C01810=1043.766,333.386,381.693,172.543,41.628,158.015
C01811=1043.756,333.058,381.740,172.537,41.623,158.014
C01812=1043.749,332.811,381.775,172.532,41.620,158.013
C01813=1043.742,332.564,381.811,172.528,41.617,158.012
C01814=1043.736,332.315,381.847,172.522,41.614,158.011
C01815=1043.728,332.069,381.883,172.518,41.611,158.010
C01816=1043.721,331.821,381.919,172.514,41.608,158.009
C01817=1043.714,331.573,381.954,172.509,41.605,158.008
C01818=1043.707,331.326,381.990,172.505,41.602,158.007
C01819=1043.700,331.078,382.025,172.500,41.599,158.006
C01820=1043.693,330.832,382.061,172.495,41.595,158.005
C01821=1043.686,330.584,382.096,172.491,41.592,158.004
C01822=1043.679,330.336,382.132,172.486,41.589,158.003
C01823=1043.672,330.090,382.167,172.482,41.586,158.002
C01824=1043.665,329.842,382.203,172.478,41.583,158.001
C01825=1043.657,329.594,382.238,172.473,41.580,158.000
C01826=1043.650,329.347,382.274,172.469,41.577,157.999
C01827=1043.643,329.100,382.308,172.465,41.573,157.998
C01828=1043.635,328.852,382.344,172.459,41.570,157.997
C01829=1043.629,328.605,382.379,172.456,41.568,157.996
C01830=1043.621,328.358,382.414,172.450,41.565,157.995
C01831=1043.614,328.110,382.449,172.446,41.562,157.994
C01832=1043.607,327.862,382.484,172.442,41.558,157.993
C01833=1043.600,327.615,382.519,172.437,41.556,157.993
C01834=1043.592,327.367,382.554,172.433,41.553,157.992
C01835=1043.585,327.120,382.589,172.429,41.550,157.991
C01836=1043.578,326.873,382.624,172.424,41.547,157.990
C01837=1043.571,326.625,382.659,172.420,41.544,157.989
C01838=1043.563,326.378,382.694,172.416,41.541,157.988
C01839=1043.556,326.130,382.729,172.411,41.538,157.987
C01840=1043.549,325.883,382.764,172.407,41.535,157.986
C01841=1043.541,325.635,382.799,172.403,41.532,157.985
C01842=1043.534,325.388,382.834,172.398,41.529,157.984
C01843=1043.527,325.141,382.869,172.393,41.526,157.983
C01844=1043.520,324.893,382.904,172.389,41.524,157.982
C01845=1043.513,324.646,382.939,172.384,41.521,157.981
C01846=1043.506,324.398,382.973,172.380,41.517,157.980
C01847=1043.498,324.151,383.008,172.376,41.515,157.980
C01848=1043.492,323.903,383.043,172.372,41.512,157.979
C01849=1043.485,323.656,383.078,172.367,41.509,157.978
C01850=1043.477,323.409,383.113,172.363,41.506,157.977
C01851=1043.471,323.161,383.147,172.359,41.503,157.976
C01852=1043.463,322.914,383.182,172.355,41.500,157.975
C01853=1043.456,322.666,383.217,172.350,41.497,157.974
C01854=1043.449,322.418,383.251,172.346,41.494,157.973
C01855=1043.442,322.171,383.286,172.342,41.492,157.972
C01856=1043.434,321.924,383.321,172.338,41.488,157.971
C01857=1043.428,321.676,383.355,172.333,41.486,157.970
C01858=1043.420,321.429,383.390,172.329,41.483,157.969
C01859=1043.414,321.181,383.425,172.325,41.480,157.969
C01860=1043.407,320.933,383.459,172.321,41.477,157.968
C01861=1043.400,320.686,383.494,172.317,41.474,157.967
C01862=1043.393,320.438,383.528,172.312,41.471,157.966
C01863=1043.386,320.191,383.563,172.308,41.469,157.965
C01864=1043.376,319.858,383.609,172.302,41.465,157.964
C01865=1043.367,319.524,383.656,172.297,41.461,157.963
C01866=1043.358,319.191,383.702,172.291,41.457,157.962
C01867=1043.348,318.858,383.749,172.285,41.453,157.960
C01868=1043.342,318.611,383.782,172.281,41.451,157.959
C01869=1043.335,318.363,383.817,172.277,41.447,157.958
C01870=1043.328,318.116,383.851,172.273,41.445,157.958
C01871=1043.321,317.868,383.886,172.268,41.442,157.957
C01872=1043.314,317.621,383.920,172.264,41.439,157.956
C01873=1043.307,317.373,383.955,172.260,41.437,157.955
C01874=1043.300,317.126,383.989,172.256,41.433,157.954
C01875=1043.293,316.878,384.024,172.252,41.431,157.953
C01876=1043.286,316.630,384.057,172.248,41.428,157.952
C01877=1043.280,316.383,384.091,172.244,41.425,157.952
C01878=1043.273,316.136,384.126,172.240,41.423,157.951
C01879=1043.266,315.888,384.160,172.236,41.419,157.950
C01880=1043.259,315.640,384.194,172.231,41.417,157.949
C01881=1043.252,315.392,384.229,172.227,41.414,157.948
C01882=1043.245,315.145,384.263,172.223,41.411,157.947
C01883=1043.239,314.898,384.297,172.219,41.409,157.946
C01884=1043.232,314.650,384.331,172.215,41.406,157.946
C01885=1043.225,314.402,384.366,172.211,41.403,157.945
C01886=1043.218,314.154,384.399,172.207,41.400,157.944
C01887=1043.212,313.908,384.434,172.204,41.398,157.943
C01888=1043.205,313.660,384.468,172.200,41.395,157.942
C01889=1043.198,313.412,384.502,172.196,41.392,157.941
C01890=1043.191,313.164,384.536,172.192,41.389,157.940
C01891=1043.185,312.917,384.570,172.188,41.387,157.940
C01892=1043.178,312.669,384.604,172.184,41.383,157.939
C01893=1043.171,312.422,384.638,172.180,41.381,157.938
C01894=1043.164,312.175,384.671,172.176,41.378,157.937
C01895=1043.157,311.927,384.705,172.171,41.376,157.936
C01896=1043.150,311.679,384.739,172.167,41.373,157.935
C01897=1043.143,311.432,384.773,172.163,41.371,157.935
C01898=1043.136,311.183,384.806,172.159,41.368,157.934
C01899=1043.129,310.936,384.839,172.155,41.365,157.933
C01900=1043.122,310.689,384.873,172.151,41.363,157.932
C01901=1043.115,310.441,384.907,172.147,41.360,157.931
C01902=1043.108,310.193,384.940,172.143,41.358,157.931
C01903=1043.101,309.946,384.973,172.140,41.355,157.930
C01904=1043.093,309.698,385.007,172.136,41.352,157.929
C01905=1043.086,309.451,385.041,172.132,41.350,157.928
C01906=1043.080,309.203,385.073,172.128,41.348,157.927
C01907=1043.073,308.955,385.107,172.124,41.345,157.927
C01908=1043.066,308.708,385.141,172.120,41.343,157.926
C01909=1043.059,308.459,385.174,172.116,41.340,157.925
C01910=1043.052,308.212,385.208,172.112,41.337,157.924
C01911=1043.044,307.965,385.241,172.108,41.335,157.923
C01912=1043.038,307.718,385.274,172.105,41.332,157.923
C01913=1043.031,307.470,385.307,172.101,41.330,157.922
C01914=1043.024,307.222,385.341,172.097,41.327,157.921
C01915=1043.017,306.975,385.374,172.093,41.325,157.920
C01916=1043.010,306.726,385.407,172.089,41.322,157.920
C01917=1043.003,306.479,385.441,172.085,41.320,157.919
C01918=1042.996,306.232,385.474,172.081,41.317,157.918
C01919=1042.989,305.984,385.507,172.077,41.314,157.917
C01920=1042.980,305.655,385.551,172.072,41.311,157.916
C01921=1042.971,305.326,385.595,172.067,41.308,157.915
C01922=1042.962,304.998,385.639,172.062,41.305,157.914
C01923=1042.953,304.669,385.683,172.057,41.302,157.913
C01924=1042.946,304.422,385.716,172.053,41.299,157.912
C01925=1042.939,304.174,385.749,172.049,41.296,157.911
C01926=1042.933,303.926,385.782,172.045,41.294,157.911
C01927=1042.925,303.679,385.815,172.041,41.291,157.910
C01928=1042.919,303.431,385.848,172.038,41.289,157.909
C01929=1042.912,303.183,385.881,172.034,41.286,157.908
C01930=1042.905,302.936,385.915,172.030,41.284,157.908
C01931=1042.898,302.688,385.948,172.026,41.281,157.907
C01932=1042.892,302.440,385.981,172.023,41.279,157.906
C01933=1042.884,302.193,386.014,172.019,41.277,157.905
C01934=1042.878,301.945,386.046,172.015,41.274,157.905
C01935=1042.871,301.697,386.079,172.011,41.271,157.904
C01936=1042.864,301.449,386.112,172.008,41.269,157.903
C01937=1042.858,301.202,386.146,172.004,41.267,157.902
C01938=1042.850,300.954,386.178,172.000,41.264,157.902
C01939=1042.844,300.707,386.211,171.996,41.261,157.901
C01940=1042.838,300.459,386.244,171.992,41.259,157.900
C01941=1042.831,300.211,386.277,171.989,41.257,157.899
C01942=1042.824,299.963,386.310,171.985,41.254,157.899
C01943=1042.816,299.716,386.343,171.982,41.252,157.898
C01944=1042.810,299.468,386.376,171.978,41.249,157.897
C01945=1042.804,299.221,386.408,171.974,41.247,157.896
C01946=1042.797,298.972,386.441,171.970,41.244,157.895
C01947=1042.791,298.725,386.474,171.967,41.242,157.895
C01948=1042.784,298.477,386.506,171.963,41.239,157.894
C01949=1042.777,298.229,386.539,171.960,41.237,157.893
C01950=1042.770,297.981,386.572,171.956,41.235,157.893
C01951=1042.764,297.734,386.605,171.952,41.232,157.892
C01952=1042.758,297.486,386.638,171.948,41.229,157.891
C01953=1042.750,297.238,386.670,171.945,41.227,157.890
C01954=1042.744,296.991,386.703,171.941,41.225,157.890
C01955=1042.738,296.743,386.736,171.938,41.223,157.889
C01956=1042.731,296.496,386.768,171.934,41.220,157.888
C01957=1042.724,296.248,386.801,171.930,41.217,157.887
C01958=1042.717,296.000,386.834,171.927,41.215,157.887
C01959=1042.711,295.752,386.866,171.923,41.213,157.886
C01960=1042.705,295.504,386.898,171.919,41.210,157.885
C01961=1042.698,295.256,386.931,171.916,41.208,157.884
C01962=1042.691,295.009,386.963,171.913,41.206,157.884
C01963=1042.684,294.761,386.996,171.909,41.203,157.883
C01964=1042.678,294.513,387.027,171.905,41.201,157.882
C01965=1042.671,294.265,387.060,171.901,41.198,157.882
C01966=1042.664,294.018,387.093,171.898,41.196,157.881
C01967=1042.658,293.770,387.125,171.895,41.194,157.880
C01968=1042.651,293.522,387.157,171.891,41.192,157.879
C01969=1042.644,293.274,387.190,171.887,41.189,157.879
C01970=1042.637,293.026,387.221,171.884,41.187,157.878
C01971=1042.630,292.779,387.253,171.881,41.185,157.877
C01972=1042.624,292.531,387.286,171.877,41.182,157.877
C01973=1042.616,292.283,387.318,171.873,41.180,157.876
C01974=1042.609,292.035,387.350,171.869,41.177,157.875
C01975=1042.603,291.787,387.382,171.866,41.175,157.875
C01976=1042.594,291.475,387.423,171.862,41.173,157.874
C01977=1042.586,291.163,387.462,171.858,41.170,157.873
C01978=1042.578,290.851,387.503,171.853,41.167,157.872
C01979=1042.569,290.539,387.544,171.849,41.164,157.871
C01980=1042.562,290.290,387.576,171.845,41.162,157.870
C01981=1042.556,290.042,387.608,171.841,41.159,157.870
C01982=1042.549,289.795,387.640,171.837,41.157,157.869
C01983=1042.542,289.547,387.671,171.835,41.155,157.868
C01984=1042.535,289.300,387.703,171.831,41.153,157.868
C01985=1042.529,289.052,387.735,171.827,41.150,157.867
C01986=1042.522,288.804,387.767,171.824,41.148,157.866
C01987=1042.515,288.556,387.799,171.821,41.146,157.866
C01988=1042.508,288.308,387.831,171.817,41.143,157.865
C01989=1042.501,288.060,387.862,171.814,41.141,157.864
C01990=1042.495,287.812,387.895,171.810,41.139,157.864
C01991=1042.488,287.564,387.926,171.807,41.137,157.863
C01992=1042.482,287.316,387.958,171.803,41.135,157.862
C01993=1042.475,287.069,387.989,171.800,41.132,157.861
C01994=1042.468,286.821,388.021,171.796,41.130,157.861
C01995=1042.461,286.573,388.053,171.793,41.128,157.860
C01996=1042.454,286.325,388.084,171.790,41.126,157.860
C01997=1042.448,286.077,388.116,171.786,41.123,157.859
C01998=1042.442,285.829,388.148,171.782,41.121,157.858
C01999=1042.434,285.581,388.179,171.780,41.119,157.857
C02000=1042.427,285.333,388.212,171.776,41.117,157.857
C02001=1042.421,285.086,388.243,171.772,41.115,157.856
C02002=1042.414,284.838,388.275,171.770,41.113,157.856
C02003=1042.407,284.590,388.306,171.766,41.110,157.855
C02004=1042.400,284.342,388.337,171.762,41.108,157.854
C02005=1042.394,284.094,388.369,171.759,41.106,157.854
C02006=1042.387,283.846,388.400,171.755,41.104,157.853
C02007=1042.380,283.598,388.432,171.752,41.102,157.852
C02008=1042.373,283.350,388.463,171.749,41.100,157.852
C02009=1042.367,283.102,388.495,171.745,41.098,157.851
C02010=1042.360,282.854,388.526,171.743,41.096,157.850
C02011=1042.353,282.607,388.557,171.739,41.093,157.850
C02012=1042.347,282.359,388.589,171.735,41.091,157.849
C02013=1042.340,282.111,388.620,171.732,41.089,157.848
C02014=1042.333,281.863,388.652,171.729,41.087,157.848
C02015=1042.326,281.615,388.683,171.726,41.084,157.847
C02016=1042.320,281.366,388.714,171.722,41.082,157.846
C02017=1042.314,281.119,388.745,171.719,41.080,157.846
C02018=1042.307,280.871,388.776,171.716,41.078,157.845
C02019=1042.300,280.623,388.808,171.712,41.076,157.844
C02020=1042.294,280.376,388.839,171.709,41.073,157.844
C02021=1042.287,280.128,388.871,171.706,41.071,157.843
C02022=1042.280,279.880,388.902,171.702,41.069,157.842
C02023=1042.274,279.631,388.933,171.699,41.067,157.842
C02024=1042.267,279.383,388.964,171.695,41.065,157.841
C02025=1042.260,279.135,388.996,171.693,41.063,157.841
C02026=1042.254,278.888,389.027,171.689,41.061,157.840
C02027=1042.248,278.640,389.057,171.686,41.059,157.839
C02028=1042.240,278.392,389.088,171.683,41.057,157.839
C02029=1042.234,278.144,389.120,171.679,41.054,157.838
C02030=1042.227,277.896,389.150,171.676,41.052,157.837
C02031=1042.220,277.648,389.182,171.673,41.050,157.837
C02032=1042.212,277.348,389.219,171.669,41.048,157.836
C02033=1042.204,277.047,389.257,171.665,41.045,157.835
C02034=1042.196,276.747,389.294,171.661,41.043,157.834
C02035=1042.187,276.446,389.331,171.657,41.040,157.834
C02036=1042.181,276.198,389.363,171.654,41.038,157.833
C02037=1042.175,275.950,389.393,171.651,41.036,157.832
C02038=1042.168,275.702,389.425,171.647,41.034,157.832
C02039=1042.161,275.454,389.455,171.644,41.032,157.831
C02040=1042.154,275.206,389.486,171.641,41.030,157.831
C02041=1042.148,274.958,389.517,171.638,41.027,157.830
C02042=1042.142,274.710,389.548,171.634,41.025,157.829
C02043=1042.135,274.462,389.578,171.632,41.023,157.829
C02044=1042.128,274.214,389.609,171.628,41.021,157.828
C02045=1042.121,273.966,389.640,171.625,41.020,157.828
C02046=1042.114,273.718,389.671,171.622,41.017,157.827
C02047=1042.108,273.470,389.701,171.619,41.015,157.826
C02048=1042.101,273.223,389.732,171.615,41.013,157.826
C02049=1042.094,272.974,389.763,171.613,41.011,157.825
C02050=1042.088,272.726,389.794,171.609,41.009,157.824
C02051=1042.081,272.479,389.824,171.606,41.007,157.824
C02052=1042.075,272.230,389.855,171.603,41.005,157.823
C02053=1042.068,271.982,389.886,171.600,41.003,157.822
C02054=1042.061,271.734,389.916,171.596,41.001,157.822
C02055=1042.055,271.486,389.947,171.594,40.999,157.821
C02056=1042.049,271.238,389.977,171.591,40.997,157.821
C02057=1042.041,270.990,390.008,171.587,40.995,157.820
C02058=1042.035,270.742,390.039,171.585,40.992,157.819
C02059=1042.028,270.494,390.069,171.581,40.990,157.819
C02060=1042.022,270.246,390.099,171.578,40.989,157.818
C02061=1042.014,269.998,390.130,171.575,40.987,157.818
C02062=1042.009,269.750,390.160,171.572,40.984,157.817
C02063=1042.001,269.502,390.191,171.568,40.982,157.816
C02064=1041.995,269.254,390.222,171.566,40.980,157.816
C02065=1041.988,269.005,390.252,171.562,40.979,157.815
C02066=1041.982,268.758,390.282,171.559,40.977,157.815
C02067=1041.975,268.509,390.312,171.557,40.974,157.814
C02068=1041.968,268.261,390.342,171.553,40.972,157.813
C02069=1041.962,268.013,390.373,171.550,40.970,157.813
C02070=1041.955,267.765,390.403,171.547,40.969,157.812
C02071=1041.949,267.517,390.433,171.544,40.966,157.812
C02072=1041.942,267.269,390.463,171.540,40.964,157.811
C02073=1041.935,267.021,390.494,171.538,40.962,157.811
C02074=1041.929,266.773,390.524,171.535,40.961,157.810
C02075=1041.921,266.525,390.554,171.531,40.959,157.809
C02076=1041.915,266.276,390.585,171.529,40.956,157.809
C02077=1041.908,266.029,390.614,171.525,40.954,157.808
C02078=1041.901,265.781,390.644,171.523,40.953,157.808
C02079=1041.895,265.532,390.675,171.520,40.950,157.807
C02080=1041.888,265.285,390.705,171.516,40.948,157.806
C02081=1041.881,265.036,390.735,171.514,40.946,157.806
C02082=1041.875,264.788,390.765,171.510,40.945,157.805
C02083=1041.868,264.540,390.795,171.507,40.943,157.805
C02084=1041.861,264.292,390.826,171.505,40.940,157.804
C02085=1041.855,264.044,390.856,171.501,40.939,157.804
C02086=1041.848,263.795,390.885,171.498,40.937,157.803
C02087=1041.842,263.548,390.915,171.496,40.934,157.802
C02088=1041.833,263.252,390.952,171.492,40.932,157.802
C02089=1041.826,262.956,390.987,171.488,40.930,157.801
C02090=1041.818,262.660,391.023,171.484,40.928,157.800
C02091=1041.810,262.364,391.059,171.481,40.925,157.800
C02092=1041.803,262.116,391.088,171.478,40.923,157.799
C02093=1041.797,261.868,391.118,171.475,40.921,157.798
C02094=1041.790,261.620,391.148,171.472,40.920,157.798
C02095=1041.783,261.372,391.177,171.469,40.917,157.797
C02096=1041.776,261.123,391.207,171.466,40.916,157.797
C02097=1041.769,260.875,391.237,171.463,40.914,157.796
C02098=1041.763,260.627,391.267,171.461,40.912,157.796
C02099=1041.756,260.379,391.297,171.457,40.910,157.795
C02100=1041.750,260.131,391.326,171.454,40.908,157.794
C02101=1041.742,259.883,391.356,171.452,40.906,157.794
C02102=1041.736,259.634,391.385,171.448,40.904,157.793
C02103=1041.729,259.386,391.415,171.445,40.903,157.793
C02104=1041.723,259.138,391.444,171.443,40.900,157.792
C02105=1041.715,258.890,391.474,171.439,40.899,157.792
C02106=1041.708,258.641,391.503,171.437,40.897,157.791
C02107=1041.701,258.394,391.533,171.434,40.895,157.791
C02108=1041.695,258.145,391.562,171.430,40.893,157.790
C02109=1041.688,257.898,391.592,171.428,40.891,157.790
C02110=1041.681,257.649,391.621,171.425,40.889,157.789
C02111=1041.675,257.401,391.651,171.422,40.888,157.788
C02112=1041.668,257.153,391.680,171.419,40.886,157.788
C02113=1041.661,256.905,391.710,171.416,40.884,157.787
C02114=1041.655,256.657,391.739,171.413,40.882,157.787
C02115=1041.648,256.408,391.769,171.410,40.880,157.786
C02116=1041.642,256.160,391.798,171.408,40.878,157.786
C02117=1041.635,255.912,391.828,171.405,40.876,157.785
C02118=1041.627,255.664,391.857,171.401,40.874,157.785
C02119=1041.621,255.415,391.886,171.399,40.872,157.784
C02120=1041.614,255.167,391.915,171.396,40.871,157.784
C02121=1041.608,254.920,391.945,171.393,40.868,157.783
C02122=1041.601,254.671,391.975,171.390,40.867,157.782
C02123=1041.595,254.423,392.004,171.387,40.865,157.782
C02124=1041.587,254.175,392.034,171.385,40.863,157.781
C02125=1041.581,253.927,392.063,171.382,40.861,157.781
C02126=1041.575,253.678,392.092,171.379,40.859,157.780
C02127=1041.568,253.430,392.121,171.376,40.857,157.780
C02128=1041.562,253.182,392.151,171.373,40.855,157.779
C02129=1041.554,252.934,392.180,171.371,40.853,157.779
C02130=1041.548,252.685,392.209,171.367,40.852,157.778
C02131=1041.541,252.437,392.238,171.365,40.850,157.777
C02132=1041.535,252.188,392.267,171.362,40.847,157.777
C02133=1041.528,251.941,392.297,171.359,40.846,157.776
C02134=1041.522,251.693,392.326,171.356,40.844,157.776
C02135=1041.515,251.444,392.356,171.353,40.842,157.775
C02136=1041.509,251.196,392.385,171.350,40.840,157.775
C02137=1041.502,250.948,392.413,171.348,40.838,157.774
C02138=1041.495,250.701,392.443,171.345,40.836,157.774
C02139=1041.488,250.452,392.472,171.342,40.835,157.773
C02140=1041.482,250.204,392.501,171.339,40.832,157.772
C02141=1041.476,249.955,392.530,171.337,40.831,157.772
C02142=1041.469,249.707,392.560,171.334,40.828,157.771
C02143=1041.463,249.458,392.589,171.331,40.827,157.771
C02144=1041.455,249.161,392.624,171.328,40.824,157.770
C02145=1041.447,248.864,392.658,171.324,40.822,157.770
C02146=1041.439,248.567,392.693,171.321,40.820,157.769
C02147=1041.431,248.269,392.728,171.318,40.818,157.768
C02148=1041.425,248.021,392.757,171.315,40.816,157.768
C02149=1041.418,247.772,392.786,171.312,40.814,157.767
C02150=1041.412,247.524,392.815,171.310,40.812,157.767
C02151=1041.406,247.276,392.844,171.307,40.810,157.766
C02152=1041.399,247.028,392.873,171.304,40.808,157.766
C02153=1041.392,246.780,392.902,171.301,40.806,157.765
C02154=1041.386,246.531,392.931,171.298,40.804,157.764
C02155=1041.380,246.283,392.960,171.296,40.802,157.764
C02156=1041.373,246.035,392.989,171.293,40.800,157.763
C02157=1041.367,245.787,393.018,171.290,40.798,157.763
C02158=1041.360,245.539,393.047,171.288,40.796,157.762
C02159=1041.353,245.290,393.076,171.285,40.794,157.762
C02160=1041.347,245.042,393.104,171.283,40.793,157.761
C02161=1041.341,244.793,393.134,171.279,40.791,157.761
C02162=1041.334,244.546,393.162,171.277,40.789,157.760
C02163=1041.328,244.298,393.191,171.274,40.787,157.759
C02164=1041.320,244.049,393.220,171.271,40.785,157.759
C02165=1041.314,243.800,393.248,171.269,40.783,157.759
C02166=1041.308,243.552,393.277,171.266,40.781,157.758
C02167=1041.301,243.304,393.306,171.264,40.780,157.757
C02168=1041.295,243.056,393.335,171.261,40.777,157.757
C02169=1041.288,242.808,393.362,171.259,40.776,157.756
C02170=1041.281,242.559,393.392,171.255,40.774,157.756
C02171=1041.275,242.311,393.421,171.252,40.772,157.755
C02172=1041.268,242.062,393.449,171.250,40.770,157.755
C02173=1041.262,241.814,393.478,171.247,40.768,157.754
C02174=1041.255,241.566,393.506,171.245,40.767,157.754
C02175=1041.249,241.318,393.534,171.242,40.764,157.753
C02176=1041.242,241.070,393.563,171.240,40.763,157.753
C02177=1041.235,240.821,393.592,171.237,40.761,157.752
C02178=1041.229,240.573,393.620,171.234,40.759,157.752
C02179=1041.222,240.324,393.649,171.232,40.757,157.751
C02180=1041.216,240.076,393.677,171.229,40.755,157.751
C02181=1041.209,239.828,393.705,171.226,40.754,157.750
C02182=1041.203,239.579,393.734,171.223,40.752,157.750
C02183=1041.196,239.332,393.762,171.221,40.750,157.749
C02184=1041.188,239.082,393.790,171.218,40.748,157.749
C02185=1041.182,238.834,393.819,171.215,40.747,157.748
C02186=1041.176,238.586,393.847,171.213,40.744,157.747
C02187=1041.169,238.338,393.875,171.210,40.743,157.747
C02188=1041.163,238.089,393.904,171.208,40.741,157.747
C02189=1041.156,237.841,393.932,171.205,40.739,157.746
C02190=1041.149,237.593,393.960,171.203,40.737,157.745
C02191=1041.143,237.345,393.989,171.200,40.736,157.745
C02192=1041.136,237.096,394.017,171.197,40.733,157.744
C02193=1041.129,236.848,394.044,171.195,40.732,157.744
C02194=1041.122,236.600,394.073,171.192,40.730,157.743
C02195=1041.116,236.351,394.101,171.190,40.728,157.743
C02196=1041.109,236.103,394.130,171.187,40.726,157.742
C02197=1041.102,235.854,394.158,171.185,40.725,157.742
C02198=1041.095,235.606,394.185,171.181,40.723,157.741
C02199=1041.089,235.358,394.214,171.179,40.721,157.741
C02200=1041.081,235.054,394.248,171.176,40.719,157.740
C02201=1041.073,234.752,394.282,171.173,40.716,157.740
C02202=1041.065,234.449,394.316,171.170,40.714,157.739
C02203=1041.057,234.146,394.351,171.167,40.712,157.738
C02204=1041.051,233.897,394.379,171.164,40.710,157.738
C02205=1041.044,233.649,394.407,171.162,40.708,157.737
C02206=1041.037,233.401,394.435,171.159,40.707,157.737
C02207=1041.031,233.152,394.463,171.157,40.704,157.736
C02208=1041.025,232.904,394.491,171.154,40.703,157.736
C02209=1041.018,232.655,394.519,171.152,40.701,157.735
C02210=1041.011,232.407,394.548,171.149,40.699,157.735
C02211=1041.004,232.159,394.575,171.147,40.697,157.734
C02212=1040.998,231.910,394.604,171.144,40.696,157.734
C02213=1040.992,231.662,394.631,171.141,40.693,157.733
C02214=1040.985,231.413,394.659,171.139,40.692,157.733
C02215=1040.978,231.165,394.687,171.136,40.690,157.732
C02216=1040.972,230.916,394.714,171.134,40.688,157.732
C02217=1040.965,230.669,394.743,171.131,40.686,157.731
C02218=1040.958,230.420,394.771,171.129,40.685,157.731
C02219=1040.951,230.172,394.798,171.126,40.682,157.730
C02220=1040.945,229.923,394.826,171.124,40.681,157.730
C02221=1040.939,229.675,394.854,171.121,40.679,157.729
C02222=1040.932,229.426,394.882,171.118,40.677,157.729
C02223=1040.925,229.178,394.910,171.116,40.675,157.728
C02224=1040.919,228.929,394.938,171.113,40.674,157.728
C02225=1040.913,228.681,394.965,171.111,40.672,157.727
C02226=1040.906,228.433,394.993,171.108,40.670,157.727
C02227=1040.899,228.185,395.020,171.106,40.668,157.726
C02228=1040.893,227.936,395.048,171.103,40.667,157.726
C02229=1040.886,227.688,395.076,171.102,40.665,157.725
C02230=1040.879,227.439,395.104,171.099,40.663,157.725
C02231=1040.872,227.191,395.131,171.097,40.661,157.724
C02232=1040.865,226.943,395.159,171.094,40.659,157.724
C02233=1040.858,226.694,395.186,171.092,40.658,157.723
C02234=1040.852,226.445,395.213,171.089,40.655,157.723
C02235=1040.845,226.197,395.241,171.086,40.654,157.722
C02236=1040.839,225.948,395.269,171.084,40.652,157.722
C02237=1040.833,225.701,395.296,171.081,40.651,157.721
C02238=1040.826,225.452,395.324,171.079,40.648,157.721
C02239=1040.818,225.204,395.351,171.076,40.647,157.720
C02240=1040.812,224.956,395.379,171.074,40.645,157.720
C02241=1040.805,224.706,395.406,171.071,40.643,157.719
C02242=1040.799,224.458,395.433,171.070,40.641,157.719
C02243=1040.792,224.210,395.461,171.067,40.639,157.718
C02244=1040.785,223.961,395.489,171.065,40.638,157.718
C02245=1040.779,223.713,395.516,171.062,40.636,157.717
C02246=1040.772,223.465,395.543,171.060,40.634,157.717
C02247=1040.766,223.216,395.570,171.057,40.632,157.716
C02248=1040.759,222.968,395.598,171.055,40.631,157.716
C02249=1040.752,222.719,395.626,171.052,40.629,157.715
C02250=1040.746,222.471,395.653,171.049,40.627,157.715
C02251=1040.740,222.223,395.680,171.048,40.625,157.714
C02252=1040.732,221.974,395.707,171.045,40.623,157.714
C02253=1040.726,221.725,395.734,171.043,40.621,157.713
C02254=1040.719,221.477,395.762,171.040,40.620,157.713
C02255=1040.713,221.229,395.789,171.038,40.618,157.712
C02256=1040.704,220.918,395.824,171.035,40.616,157.712
C02257=1040.697,220.608,395.858,171.032,40.613,157.711
C02258=1040.688,220.297,395.892,171.029,40.611,157.711
C02259=1040.680,219.987,395.926,171.026,40.608,157.710
C02260=1040.674,219.738,395.953,171.024,40.607,157.709
C02261=1040.666,219.490,395.980,171.021,40.605,157.709
C02262=1040.660,219.240,396.007,171.019,40.603,157.708
C02263=1040.653,218.992,396.035,171.017,40.602,157.708
C02264=1040.647,218.745,396.061,171.015,40.600,157.708
C02265=1040.640,218.496,396.088,171.012,40.598,157.707
C02266=1040.633,218.247,396.116,171.009,40.596,157.706
C02267=1040.626,217.998,396.143,171.007,40.595,157.706
C02268=1040.620,217.751,396.169,171.004,40.593,157.706
C02269=1040.613,217.502,396.196,171.003,40.591,157.705
C02270=1040.607,217.253,396.223,171.000,40.589,157.705
C02271=1040.599,217.005,396.251,170.998,40.587,157.704
C02272=1040.594,216.756,396.277,170.995,40.586,157.704
C02273=1040.586,216.508,396.304,170.993,40.584,157.703
C02274=1040.580,216.259,396.331,170.991,40.582,157.703
C02275=1040.572,216.011,396.358,170.989,40.580,157.702
C02276=1040.567,215.763,396.385,170.986,40.578,157.702
C02277=1040.560,215.514,396.412,170.984,40.577,157.701
C02278=1040.553,215.265,396.439,170.981,40.575,157.701
C02279=1040.547,215.017,396.466,170.980,40.573,157.700
C02280=1040.540,214.769,396.493,170.977,40.571,157.700
C02281=1040.533,214.520,396.520,170.975,40.569,157.699
C02282=1040.527,214.272,396.546,170.972,40.568,157.699
C02283=1040.520,214.023,396.574,170.969,40.566,157.698
C02284=1040.513,213.775,396.600,170.968,40.564,157.698
C02285=1040.507,213.526,396.627,170.965,40.562,157.697
C02286=1040.500,213.278,396.655,170.963,40.561,157.697
C02287=1040.493,213.029,396.681,170.960,40.558,157.696
C02288=1040.488,212.781,396.708,170.959,40.557,157.696
C02289=1040.480,212.533,396.735,170.956,40.555,157.695
C02290=1040.474,212.284,396.762,170.954,40.553,157.695
C02291=1040.467,212.035,396.788,170.951,40.551,157.694
C02292=1040.461,211.786,396.815,170.950,40.549,157.694
C02293=1040.454,211.539,396.842,170.947,40.548,157.693
C02294=1040.448,211.290,396.869,170.945,40.546,157.693
C02295=1040.441,211.041,396.895,170.942,40.544,157.692
C02296=1040.434,210.793,396.921,170.941,40.542,157.692
C02297=1040.428,210.544,396.948,170.938,40.540,157.691
C02298=1040.420,210.296,396.975,170.936,40.539,157.691
C02299=1040.415,210.048,397.002,170.933,40.537,157.691
C02300=1040.407,209.799,397.028,170.932,40.535,157.690
C02301=1040.401,209.551,397.054,170.929,40.533,157.689
C02302=1040.395,209.302,397.081,170.927,40.531,157.689
C02303=1040.387,209.053,397.108,170.925,40.530,157.689
C02304=1040.381,208.805,397.134,170.923,40.528,157.688
C02305=1040.375,208.556,397.161,170.920,40.526,157.688
C02306=1040.368,208.308,397.187,170.918,40.524,157.687
C02307=1040.361,208.060,397.214,170.916,40.522,157.687
C02308=1040.353,207.811,397.241,170.914,40.521,157.686
C02309=1040.348,207.563,397.267,170.911,40.519,157.686
C02310=1040.341,207.314,397.294,170.909,40.517,157.685
C02311=1040.334,207.066,397.320,170.907,40.515,157.685
C02312=1040.326,206.760,397.352,170.904,40.513,157.684
C02313=1040.318,206.455,397.384,170.902,40.510,157.684
C02314=1040.310,206.150,397.417,170.899,40.509,157.683
C02315=1040.301,205.845,397.449,170.896,40.507,157.682
C02316=1040.275,204.794,397.555,170.609,40.403,157.648
C02317=1040.269,204.545,397.581,170.606,40.402,157.648
C02318=1040.263,204.296,397.606,170.602,40.401,157.647
C02319=1040.256,204.048,397.631,170.599,40.400,157.647
C02320=1040.250,203.799,397.657,170.597,40.399,157.647
C02321=1040.245,203.551,397.682,170.593,40.397,157.646
C02322=1040.239,203.302,397.706,170.590,40.397,157.646
C02323=1040.233,203.053,397.732,170.587,40.395,157.646
C02324=1040.226,202.805,397.756,170.584,40.395,157.645
C02325=1040.219,202.556,397.782,170.581,40.394,157.645
C02326=1040.213,202.307,397.807,170.578,40.393,157.645
C02327=1040.208,202.059,397.831,170.575,40.392,157.644
C02328=1040.202,201.810,397.857,170.572,40.391,157.644
C02329=1040.195,201.561,397.882,170.569,40.390,157.644
C02330=1040.189,201.313,397.907,170.566,40.388,157.643
C02331=1040.183,201.063,397.932,170.563,40.387,157.643
C02332=1040.176,200.815,397.957,170.560,40.386,157.643
C02333=1040.170,200.566,397.982,170.557,40.385,157.642
C02334=1040.165,200.318,398.006,170.554,40.385,157.642
C02335=1040.158,200.069,398.031,170.551,40.384,157.642
C02336=1040.152,199.820,398.056,170.548,40.383,157.641
C02337=1040.145,199.572,398.080,170.545,40.382,157.641
C02338=1040.139,199.323,398.105,170.542,40.381,157.641
C02339=1040.133,199.074,398.130,170.539,40.380,157.640
C02340=1040.127,198.826,398.154,170.536,40.379,157.640
C02341=1040.121,198.577,398.179,170.533,40.378,157.640
C02342=1040.114,198.329,398.204,170.530,40.377,157.639
C02343=1040.108,198.079,398.229,170.527,40.377,157.639
C02344=1040.101,197.831,398.253,170.525,40.376,157.639
C02345=1040.096,197.582,398.278,170.521,40.375,157.638
C02346=1040.090,197.333,398.302,170.518,40.374,157.638
C02347=1040.083,197.085,398.327,170.516,40.373,157.638
C02348=1040.077,196.835,398.352,170.512,40.372,157.637
C02349=1040.070,196.587,398.376,170.510,40.371,157.637
C02350=1040.065,196.338,398.401,170.507,40.370,157.637
C02351=1040.058,196.090,398.425,170.503,40.370,157.637
C02352=1040.052,195.841,398.450,170.501,40.368,157.636
C02353=1040.046,195.593,398.474,170.498,40.368,157.636
C02354=1040.040,195.344,398.499,170.494,40.367,157.636
C02355=1040.033,195.095,398.523,170.492,40.366,157.635
C02356=1040.027,194.846,398.548,170.489,40.365,157.635
C02357=1040.021,194.598,398.573,170.487,40.364,157.635
C02358=1040.015,194.349,398.597,170.483,40.363,157.634
C02359=1040.009,194.100,398.622,170.480,40.362,157.634
C02360=1040.003,193.852,398.646,170.478,40.361,157.634
C02361=1039.997,193.602,398.670,170.474,40.360,157.633
C02362=1039.990,193.354,398.695,170.472,40.360,157.633
C02363=1039.984,193.105,398.719,170.469,40.359,157.633
C02364=1039.978,192.856,398.743,170.466,40.358,157.633
C02365=1039.972,192.607,398.768,170.463,40.357,157.632
C02366=1039.966,192.360,398.792,170.460,40.356,157.632
C02367=1039.960,192.110,398.817,170.458,40.356,157.632
C02368=1039.953,191.861,398.841,170.454,40.355,157.631
C02369=1039.948,191.613,398.865,170.452,40.354,157.631
C02370=1039.941,191.364,398.890,170.449,40.353,157.631
C02371=1039.935,191.116,398.914,170.445,40.352,157.630
C02372=1039.929,190.867,398.938,170.443,40.351,157.630
C02373=1039.923,190.617,398.963,170.440,40.350,157.630
C02374=1039.918,190.369,398.987,170.438,40.349,157.630
C02375=1039.911,190.121,399.012,170.434,40.348,157.629
C02376=1039.905,189.872,399.036,170.432,40.348,157.629
C02377=1039.898,189.587,399.064,170.429,40.347,157.629
C02378=1039.891,189.303,399.092,170.425,40.346,157.628
C02379=1039.884,189.018,399.119,170.422,40.345,157.628
C02380=1039.877,188.734,399.147,170.419,40.344,157.628
C02381=1039.871,188.485,399.171,170.416,40.343,157.627
C02382=1039.865,188.237,399.195,170.413,40.342,157.627
C02383=1039.859,187.988,399.220,170.411,40.341,157.627
C02384=1039.853,187.739,399.243,170.408,40.341,157.627
C02385=1039.847,187.490,399.268,170.405,40.340,157.626
C02386=1039.841,187.242,399.292,170.402,40.339,157.626
C02387=1039.835,186.992,399.316,170.400,40.338,157.626
C02388=1039.829,186.744,399.340,170.396,40.337,157.625
C02389=1039.824,186.495,399.364,170.394,40.336,157.625
C02390=1039.817,186.247,399.388,170.391,40.335,157.625
C02391=1039.812,185.997,399.413,170.388,40.334,157.624
C02392=1039.806,185.749,399.436,170.385,40.334,157.624
C02393=1039.799,185.500,399.460,170.383,40.333,157.624
C02394=1039.794,185.252,399.485,170.380,40.332,157.624
C02395=1039.787,185.003,399.509,170.377,40.332,157.623
C02396=1039.782,184.754,399.533,170.374,40.331,157.623
C02397=1039.775,184.505,399.557,170.372,40.330,157.623
C02398=1039.770,184.256,399.581,170.369,40.329,157.622
C02399=1039.764,184.008,399.605,170.366,40.328,157.622
C02400=1039.758,183.759,399.629,170.363,40.327,157.622
C02401=1039.752,183.511,399.653,170.361,40.326,157.622
C02402=1039.745,183.261,399.676,170.358,40.326,157.621
C02403=1039.739,183.013,399.700,170.355,40.325,157.621
C02404=1039.733,182.764,399.724,170.352,40.325,157.621
C02405=1039.727,182.515,399.748,170.350,40.324,157.621
C02406=1039.720,182.266,399.771,170.347,40.323,157.620
C02407=1039.714,182.018,399.795,170.344,40.323,157.620
C02408=1039.708,181.769,399.819,170.341,40.322,157.620
C02409=1039.702,181.520,399.842,170.339,40.321,157.620
C02410=1039.695,181.271,399.865,170.336,40.321,157.619
C02411=1039.689,181.023,399.889,170.333,40.320,157.619
C02412=1039.682,180.773,399.912,170.330,40.320,157.619
C02413=1039.676,180.525,399.936,170.328,40.319,157.619
C02414=1039.670,180.276,399.960,170.325,40.318,157.618
C02415=1039.664,180.027,399.983,170.323,40.318,157.618
C02416=1039.657,179.778,400.007,170.319,40.317,157.618
C02417=1039.651,179.529,400.030,170.317,40.316,157.618
C02418=1039.645,179.280,400.054,170.314,40.316,157.618
C02419=1039.639,179.032,400.077,170.312,40.315,157.617
C02420=1039.632,178.783,400.100,170.308,40.315,157.617
C02421=1039.626,178.534,400.124,170.306,40.314,157.617
C02422=1039.620,178.285,400.147,170.303,40.313,157.617
C02423=1039.613,178.036,400.171,170.301,40.313,157.616
C02424=1039.608,177.788,400.194,170.297,40.313,157.616
C02425=1039.601,177.539,400.218,170.295,40.312,157.616
C02426=1039.595,177.290,400.241,170.292,40.311,157.616
C02427=1039.589,177.041,400.264,170.290,40.310,157.615
C02428=1039.583,176.792,400.288,170.288,40.310,157.615
C02429=1039.576,176.544,400.311,170.284,40.309,157.615
C02430=1039.570,176.294,400.334,170.282,40.308,157.615
C02431=1039.564,176.046,400.358,170.279,40.308,157.614
C02432=1039.558,175.797,400.381,170.277,40.308,157.614
C02433=1039.551,175.548,400.405,170.273,40.307,157.614
C02434=1039.546,175.299,400.428,170.271,40.306,157.614
C02435=1039.540,175.050,400.451,170.268,40.306,157.614
C02436=1039.533,174.801,400.475,170.266,40.305,157.613
C02437=1039.527,174.553,400.497,170.264,40.304,157.613
C02438=1039.521,174.304,400.521,170.260,40.304,157.613
C02439=1039.514,174.055,400.544,170.258,40.303,157.613
C02440=1039.509,173.806,400.567,170.255,40.303,157.612
C02441=1039.502,173.521,400.594,170.253,40.302,157.612
C02442=1039.495,173.237,400.620,170.249,40.301,157.612
C02443=1039.488,172.952,400.647,170.246,40.301,157.612
C02444=1039.481,172.667,400.673,170.243,40.300,157.611
C02445=1039.474,172.418,400.697,170.241,40.300,157.611
C02446=1039.468,172.169,400.720,170.238,40.299,157.611
C02447=1039.463,171.921,400.743,170.235,40.298,157.611
C02448=1039.456,171.672,400.765,170.233,40.298,157.610
C02449=1039.450,171.423,400.789,170.230,40.297,157.610
C02450=1039.444,171.174,400.812,170.227,40.296,157.610
C02451=1039.438,170.925,400.835,170.225,40.296,157.610
C02452=1039.432,170.676,400.858,170.222,40.295,157.609
C02453=1039.426,170.427,400.882,170.220,40.295,157.609
C02454=1039.420,170.178,400.905,170.217,40.294,157.609
C02455=1039.414,169.930,400.927,170.214,40.294,157.609
C02456=1039.408,169.681,400.950,170.212,40.293,157.608
C02457=1039.401,169.432,400.974,170.209,40.293,157.608
C02458=1039.395,169.183,400.997,170.207,40.292,157.608
C02459=1039.390,168.934,401.020,170.205,40.291,157.608
C02460=1039.383,168.686,401.043,170.201,40.291,157.608
C02461=1039.378,168.437,401.066,170.199,40.290,157.607
C02462=1039.371,168.188,401.089,170.197,40.289,157.607
C02463=1039.365,167.939,401.113,170.194,40.289,157.607
C02464=1039.359,167.690,401.136,170.191,40.288,157.607
C02465=1039.354,167.441,401.158,170.189,40.288,157.607
C02466=1039.347,167.192,401.181,170.186,40.287,157.606
C02467=1039.342,166.944,401.204,170.184,40.287,157.606
C02468=1039.336,166.695,401.227,170.182,40.286,157.606
C02469=1039.329,166.445,401.250,170.178,40.285,157.605
C02470=1039.324,166.196,401.273,170.176,40.285,157.605
C02471=1039.317,165.948,401.296,170.174,40.284,157.605
C02472=1039.311,165.699,401.319,170.171,40.283,157.605
C02473=1039.305,165.450,401.342,170.169,40.283,157.605
C02474=1039.300,165.201,401.365,170.166,40.283,157.604
C02475=1039.294,164.953,401.388,170.163,40.282,157.604
C02476=1039.288,164.704,401.410,170.161,40.281,157.604
C02477=1039.282,164.455,401.433,170.159,40.281,157.604
C02478=1039.275,164.205,401.456,170.155,40.280,157.604
C02479=1039.270,163.957,401.479,170.153,40.279,157.603
C02480=1039.264,163.708,401.502,170.151,40.279,157.603
C02481=1039.258,163.459,401.525,170.149,40.279,157.603
C02482=1039.252,163.210,401.548,170.146,40.278,157.603
C02483=1039.246,162.961,401.571,170.143,40.277,157.602
C02484=1039.240,162.712,401.594,170.141,40.277,157.602
C02485=1039.234,162.464,401.616,170.138,40.276,157.602
C02486=1039.228,162.215,401.639,170.136,40.275,157.602
C02487=1039.222,161.966,401.662,170.134,40.275,157.601
C02488=1039.217,161.717,401.685,170.131,40.274,157.601
C02489=1039.211,161.468,401.707,170.128,40.274,157.601
C02490=1039.205,161.219,401.729,170.126,40.273,157.601
C02491=1039.199,160.970,401.752,170.124,40.273,157.601
C02492=1039.193,160.721,401.775,170.122,40.272,157.600
C02493=1039.188,160.472,401.798,170.118,40.272,157.600
C02494=1039.181,160.224,401.820,170.116,40.271,157.600
C02495=1039.175,159.975,401.843,170.114,40.270,157.600
C02496=1039.169,159.726,401.865,170.111,40.270,157.600
C02497=1039.164,159.477,401.888,170.109,40.270,157.599
C02498=1039.157,159.228,401.910,170.106,40.269,157.599
C02499=1039.151,158.979,401.933,170.104,40.269,157.599
C02500=1039.145,158.729,401.955,170.101,40.268,157.599
C02501=1039.138,158.481,401.978,170.099,40.268,157.599
C02502=1039.132,158.232,402.001,170.097,40.268,157.598
C02503=1039.126,157.983,402.022,170.093,40.267,157.598
C02504=1039.120,157.734,402.045,170.091,40.267,157.598
C02505=1039.113,157.449,402.070,170.088,40.266,157.598
C02506=1039.106,157.164,402.096,170.086,40.265,157.598
C02507=1039.100,156.878,402.121,170.083,40.265,157.597
C02508=1039.092,156.593,402.147,170.080,40.265,157.597
C02509=1039.086,156.345,402.170,170.077,40.264,157.597
C02510=1039.080,156.096,402.191,170.075,40.264,157.597
C02511=1039.074,155.847,402.214,170.073,40.263,157.597
C02512=1039.068,155.597,402.236,170.070,40.263,157.596
C02513=1039.062,155.349,402.259,170.068,40.263,157.596
C02514=1039.056,155.100,402.281,170.065,40.262,157.596
C02515=1039.049,154.851,402.303,170.063,40.262,157.596
C02516=1039.044,154.602,402.326,170.060,40.261,157.596
C02517=1039.038,154.353,402.347,170.058,40.260,157.595
C02518=1039.031,154.104,402.370,170.056,40.260,157.595
C02519=1039.025,153.855,402.391,170.053,40.259,157.595
C02520=1039.019,153.606,402.414,170.050,40.259,157.595
C02521=1039.013,153.357,402.436,170.048,40.259,157.595
C02522=1039.007,153.108,402.458,170.046,40.259,157.595
C02523=1039.000,152.859,402.480,170.044,40.258,157.594
C02524=1038.994,152.610,402.502,170.041,40.258,157.594
C02525=1038.989,152.361,402.524,170.039,40.258,157.594
C02526=1038.982,152.112,402.547,170.036,40.257,157.594
C02527=1038.976,151.864,402.568,170.034,40.257,157.594
C02528=1038.970,151.615,402.590,170.031,40.257,157.593
C02529=1038.964,151.366,402.612,170.029,40.256,157.593
C02530=1038.958,151.116,402.634,170.027,40.256,157.593
C02531=1038.952,150.868,402.657,170.025,40.255,157.593
C02532=1038.946,150.619,402.678,170.021,40.255,157.593
C02533=1038.939,150.370,402.701,170.019,40.254,157.593
C02534=1038.933,150.121,402.722,170.017,40.254,157.592
C02535=1038.928,149.871,402.744,170.015,40.254,157.592
C02536=1038.921,149.623,402.767,170.012,40.253,157.592
C02537=1038.915,149.374,402.788,170.010,40.253,157.592
C02538=1038.910,149.125,402.810,170.007,40.252,157.592
C02539=1038.903,148.876,402.832,170.005,40.252,157.591
C02540=1038.897,148.627,402.854,170.003,40.252,157.591
C02541=1038.891,148.378,402.875,170.000,40.251,157.591
C02542=1038.885,148.129,402.898,169.998,40.251,157.591
C02543=1038.879,147.880,402.920,169.996,40.250,157.591
C02544=1038.873,147.631,402.942,169.993,40.250,157.591
C02545=1038.867,147.382,402.963,169.990,40.250,157.590
C02546=1038.861,147.134,402.985,169.988,40.250,157.590
C02547=1038.854,146.884,403.007,169.986,40.249,157.590
C02548=1038.848,146.635,403.028,169.984,40.249,157.590
C02549=1038.842,146.386,403.050,169.982,40.248,157.590
C02550=1038.836,146.137,403.072,169.978,40.248,157.590
C02551=1038.830,145.888,403.094,169.976,40.248,157.589
C02552=1038.823,145.639,403.116,169.974,40.247,157.589
C02553=1038.818,145.391,403.137,169.972,40.247,157.589
C02554=1038.812,145.141,403.159,169.969,40.247,157.589
C02555=1038.805,144.892,403.180,169.967,40.247,157.589
C02556=1038.799,144.643,403.201,169.965,40.246,157.589
C02557=1038.792,144.394,403.223,169.962,40.246,157.588
C02558=1038.786,144.145,403.245,169.960,40.245,157.588
C02559=1038.780,143.897,403.267,169.957,40.245,157.588
C02560=1038.774,143.648,403.288,169.955,40.245,157.588
C02561=1038.768,143.399,403.310,169.953,40.245,157.588
C02562=1038.762,143.149,403.331,169.951,40.244,157.588
C02563=1038.756,142.900,403.353,169.949,40.244,157.587
C02564=1038.750,142.652,403.374,169.945,40.244,157.587
C02565=1038.744,142.402,403.396,169.943,40.243,157.587
C02566=1038.738,142.153,403.418,169.941,40.243,157.587
C02567=1038.732,141.904,403.439,169.939,40.243,157.587
C02568=1038.726,141.655,403.461,169.937,40.242,157.587
C02569=1038.718,141.370,403.485,169.934,40.242,157.586
C02570=1038.712,141.085,403.510,169.932,40.242,157.586
C02571=1038.705,140.799,403.535,169.928,40.241,157.586
C02572=1038.697,140.514,403.559,169.926,40.241,157.586
C02573=1038.691,140.265,403.581,169.924,40.240,157.586
C02574=1038.685,140.015,403.602,169.921,40.240,157.586
C02575=1038.679,139.766,403.624,169.919,40.240,157.585
C02576=1038.673,139.518,403.645,169.917,40.239,157.585
C02577=1038.667,139.268,403.667,169.915,40.239,157.585
C02578=1038.661,139.019,403.688,169.912,40.239,157.585
C02579=1038.654,138.770,403.709,169.910,40.239,157.585
C02580=1038.649,138.521,403.730,169.907,40.238,157.585
C02581=1038.643,138.272,403.752,169.905,40.238,157.585
C02582=1038.637,138.023,403.774,169.903,40.238,157.584
C02583=1038.630,137.774,403.795,169.901,40.238,157.584
C02584=1038.624,137.525,403.816,169.898,40.237,157.584
C02585=1038.618,137.276,403.837,169.896,40.237,157.584
C02586=1038.612,137.026,403.858,169.893,40.237,157.584
C02587=1038.606,136.778,403.879,169.891,40.237,157.584
C02588=1038.600,136.529,403.901,169.889,40.236,157.583
C02589=1038.593,136.280,403.922,169.887,40.236,157.583
C02590=1038.587,136.031,403.943,169.885,40.236,157.583
C02591=1038.581,135.782,403.964,169.883,40.235,157.583
C02592=1038.575,135.533,403.986,169.879,40.235,157.583
C02593=1038.568,135.284,404.007,169.877,40.235,157.583
C02594=1038.563,135.035,404.028,169.875,40.235,157.583
C02595=1038.557,134.786,404.050,169.873,40.234,157.582
C02596=1038.550,134.536,404.070,169.871,40.234,157.582
C02597=1038.544,134.288,404.091,169.869,40.234,157.582
C02598=1038.538,134.039,404.113,169.866,40.234,157.582
C02599=1038.531,133.790,404.134,169.864,40.233,157.582
C02600=1038.526,133.541,404.154,169.861,40.233,157.582
C02601=1038.520,133.291,404.176,169.859,40.233,157.581
C02602=1038.513,133.043,404.197,169.857,40.233,157.581
C02603=1038.508,132.793,404.218,169.855,40.232,157.581
C02604=1038.501,132.545,404.239,169.853,40.232,157.581
C02605=1038.495,132.296,404.260,169.850,40.231,157.581
C02606=1038.489,132.046,404.281,169.848,40.232,157.581
C02607=1038.483,131.797,404.302,169.845,40.231,157.581
C02608=1038.477,131.549,404.323,169.843,40.231,157.580
C02609=1038.471,131.299,404.344,169.841,40.230,157.580
C02610=1038.464,131.050,404.365,169.839,40.231,157.580
C02611=1038.459,130.801,404.386,169.837,40.230,157.580
C02612=1038.452,130.552,404.407,169.835,40.230,157.580
C02613=1038.445,130.303,404.428,169.832,40.230,157.580
C02614=1038.440,130.054,404.448,169.830,40.230,157.580
C02615=1038.433,129.805,404.469,169.828,40.230,157.580
C02616=1038.427,129.555,404.490,169.825,40.229,157.579
C02617=1038.421,129.307,404.511,169.823,40.229,157.579
C02618=1038.414,129.058,404.531,169.821,40.229,157.579
C02619=1038.409,128.809,404.552,169.818,40.229,157.579
C02620=1038.402,128.560,404.573,169.816,40.229,157.579
C02621=1038.395,128.310,404.593,169.814,40.228,157.579
C02622=1038.390,128.062,404.614,169.812,40.229,157.579
C02623=1038.383,127.812,404.635,169.810,40.228,157.579
C02624=1038.376,127.563,404.656,169.808,40.228,157.578
C02625=1038.371,127.314,404.676,169.805,40.228,157.578
C02626=1038.364,127.065,404.697,169.802,40.228,157.578
C02627=1038.358,126.816,404.717,169.800,40.228,157.578
C02628=1038.351,126.567,404.738,169.798,40.227,157.578
C02629=1038.346,126.318,404.759,169.796,40.227,157.578
C02630=1038.340,126.069,404.779,169.794,40.227,157.578
C02631=1038.333,125.820,404.800,169.792,40.227,157.577
C02632=1038.327,125.571,404.821,169.790,40.226,157.577
C02633=1038.320,125.285,404.845,169.787,40.227,157.577
C02634=1038.313,124.999,404.869,169.784,40.226,157.577
C02635=1038.306,124.714,404.892,169.781,40.226,157.577
C02636=1038.299,124.428,404.915,169.779,40.226,157.577
C02637=1038.292,124.179,404.936,169.777,40.226,157.577
C02638=1038.286,123.929,404.956,169.775,40.225,157.576
C02639=1038.280,123.680,404.977,169.773,40.225,157.576
C02640=1038.273,123.431,404.998,169.770,40.225,157.576
C02641=1038.267,123.183,405.018,169.768,40.225,157.576
C02642=1038.262,122.933,405.039,169.766,40.225,157.576
C02643=1038.255,122.685,405.060,169.763,40.224,157.576
C02644=1038.249,122.435,405.080,169.761,40.224,157.576
C02645=1038.243,122.186,405.100,169.759,40.224,157.576
C02646=1038.237,121.936,405.121,169.757,40.224,157.575
C02647=1038.230,121.688,405.141,169.755,40.224,157.575
C02648=1038.224,121.439,405.162,169.753,40.223,157.575
C02649=1038.219,121.190,405.182,169.751,40.224,157.575
C02650=1038.212,120.940,405.203,169.748,40.223,157.575
C02651=1038.206,120.692,405.223,169.745,40.223,157.575
C02652=1038.200,120.443,405.244,169.743,40.223,157.575
C02653=1038.194,120.193,405.264,169.741,40.223,157.575
C02654=1038.188,119.944,405.284,169.739,40.222,157.574
C02655=1038.181,119.696,405.305,169.737,40.222,157.574
C02656=1038.176,119.446,405.326,169.735,40.222,157.574
C02657=1038.169,119.197,405.346,169.733,40.222,157.574
C02658=1038.163,118.948,405.366,169.731,40.222,157.574
C02659=1038.157,118.698,405.387,169.729,40.221,157.574
C02660=1038.151,118.450,405.407,169.727,40.221,157.574
C02661=1038.145,118.201,405.428,169.724,40.221,157.573
C02662=1038.138,117.952,405.448,169.722,40.220,157.573
C02663=1038.133,117.703,405.469,169.720,40.221,157.573
C02664=1038.127,117.453,405.489,169.717,40.220,157.573
C02665=1038.121,117.204,405.509,169.715,40.220,157.573
C02666=1038.115,116.956,405.529,169.713,40.220,157.573
C02667=1038.109,116.706,405.550,169.711,40.220,157.573
C02668=1038.103,116.457,405.570,169.708,40.219,157.572
C02669=1038.096,116.208,405.591,169.706,40.219,157.572
C02670=1038.091,115.959,405.611,169.704,40.219,157.572
C02671=1038.085,115.710,405.631,169.702,40.218,157.572
C02672=1038.078,115.461,405.652,169.700,40.219,157.572
C02673=1038.072,115.212,405.671,169.698,40.218,157.572
C02674=1038.067,114.963,405.692,169.696,40.218,157.572
C02675=1038.060,114.713,405.712,169.694,40.218,157.572
C02676=1038.054,114.464,405.732,169.692,40.218,157.571
C02677=1038.048,114.215,405.752,169.689,40.217,157.571
C02678=1038.042,113.966,405.773,169.687,40.217,157.571
C02679=1038.036,113.717,405.793,169.685,40.217,157.571
C02680=1038.030,113.468,405.813,169.683,40.216,157.571
C02681=1038.024,113.219,405.833,169.681,40.217,157.571
C02682=1038.018,112.970,405.853,169.679,40.216,157.571
C02683=1038.012,112.721,405.873,169.676,40.216,157.571
C02684=1038.005,112.471,405.894,169.674,40.216,157.570
C02685=1037.999,112.223,405.914,169.672,40.216,157.570
C02686=1037.993,111.973,405.934,169.669,40.216,157.570
C02687=1037.987,111.724,405.954,169.667,40.216,157.570
C02688=1037.981,111.475,405.973,169.665,40.216,157.570
C02689=1037.974,111.225,405.994,169.663,40.216,157.570
C02690=1037.968,110.976,406.013,169.661,40.215,157.570
C02691=1037.962,110.728,406.033,169.659,40.215,157.570
C02692=1037.956,110.478,406.054,169.657,40.215,157.570
C02693=1037.950,110.229,406.074,169.655,40.215,157.569
C02694=1037.944,109.980,406.093,169.653,40.215,157.569
C02695=1037.937,109.730,406.113,169.651,40.215,157.569
C02696=1037.931,109.482,406.133,169.649,40.215,157.569
C02697=1037.924,109.196,406.156,169.646,40.215,157.569
C02698=1037.917,108.910,406.178,169.643,40.214,157.569
C02699=1037.910,108.624,406.201,169.640,40.215,157.569
C02700=1037.902,108.338,406.224,169.638,40.214,157.569
C02701=1037.896,108.089,406.244,169.636,40.214,157.569
C02702=1037.890,107.840,406.263,169.634,40.214,157.568
C02703=1037.884,107.591,406.283,169.632,40.214,157.568
C02704=1037.878,107.341,406.303,169.630,40.214,157.568
C02705=1037.872,107.092,406.323,169.628,40.214,157.568
C02706=1037.865,106.844,406.342,169.626,40.213,157.568
C02707=1037.858,106.594,406.362,169.624,40.214,157.568
C02708=1037.853,106.345,406.382,169.621,40.213,157.568
C02709=1037.847,106.096,406.402,169.619,40.213,157.568
C02710=1037.841,105.847,406.421,169.617,40.213,157.567
C02711=1037.833,105.597,406.441,169.614,40.213,157.567
C02712=1037.827,105.349,406.461,169.612,40.213,157.567
C02713=1037.822,105.099,406.480,169.610,40.213,157.567
C02714=1037.815,104.850,406.500,169.608,40.213,157.567
C02715=1037.809,104.601,406.520,169.606,40.213,157.567
C02716=1037.803,104.352,406.539,169.604,40.212,157.567
C02717=1037.797,104.103,406.559,169.602,40.213,157.567
C02718=1037.791,103.854,406.579,169.599,40.212,157.567
C02719=1037.785,103.604,406.599,169.597,40.212,157.566
C02720=1037.779,103.355,406.618,169.595,40.212,157.566
C02721=1037.772,103.106,406.637,169.593,40.212,157.566
C02722=1037.766,102.857,406.657,169.591,40.212,157.566
C02723=1037.760,102.608,406.677,169.589,40.212,157.566
C02724=1037.754,102.358,406.697,169.587,40.211,157.566
C02725=1037.748,102.109,406.717,169.585,40.212,157.566
C02726=1037.741,101.860,406.735,169.583,40.211,157.566
C02727=1037.735,101.612,406.755,169.581,40.211,157.566
C02728=1037.729,101.361,406.775,169.579,40.211,157.565
C02729=1037.723,101.113,406.795,169.577,40.211,157.565
C02730=1037.717,100.863,406.813,169.574,40.211,157.565
C02731=1037.711,100.615,406.833,169.572,40.211,157.565
C02732=1037.705,100.366,406.853,169.570,40.210,157.565
C02733=1037.699,100.116,406.873,169.568,40.211,157.565
C02734=1037.692,99.867,406.892,169.566,40.210,157.565
C02735=1037.686,99.618,406.912,169.564,40.210,157.565
C02736=1037.680,99.369,406.930,169.562,40.210,157.564
C02737=1037.674,99.120,406.950,169.559,40.210,157.564
C02738=1037.667,98.871,406.969,169.557,40.210,157.564
C02739=1037.661,98.621,406.989,169.555,40.210,157.564
C02740=1037.654,98.372,407.008,169.553,40.210,157.564
C02741=1037.648,98.123,407.027,169.551,40.210,157.564
C02742=1037.642,97.874,407.046,169.548,40.210,157.564
C02743=1037.636,97.625,407.066,169.546,40.210,157.564
C02744=1037.629,97.375,407.085,169.544,40.210,157.564
C02745=1037.623,97.126,407.105,169.542,40.210,157.564
C02746=1037.617,96.877,407.123,169.540,40.210,157.564
C02747=1037.611,96.628,407.143,169.538,40.210,157.563
C02748=1037.605,96.379,407.162,169.536,40.210,157.563
C02749=1037.598,96.130,407.181,169.534,40.209,157.563
C02750=1037.593,95.880,407.200,169.532,40.209,157.563
C02751=1037.585,95.631,407.220,169.530,40.210,157.563
C02752=1037.580,95.382,407.239,169.528,40.209,157.563
C02753=1037.573,95.132,407.258,169.526,40.209,157.563
C02754=1037.567,94.884,407.278,169.523,40.209,157.563
C02755=1037.561,94.634,407.297,169.521,40.209,157.563
C02756=1037.555,94.385,407.316,169.519,40.209,157.562
C02757=1037.549,94.136,407.335,169.517,40.209,157.562
C02758=1037.543,93.887,407.354,169.515,40.209,157.562
C02759=1037.536,93.637,407.373,169.513,40.209,157.562
C02760=1037.530,93.388,407.393,169.511,40.209,157.562
C02761=1037.523,93.103,407.415,169.508,40.209,157.562
C02762=1037.516,92.817,407.436,169.506,40.209,157.562
C02763=1037.509,92.531,407.459,169.504,40.208,157.562
C02764=1037.502,92.244,407.480,169.501,40.209,157.562
C02765=1037.495,91.995,407.499,169.498,40.208,157.561
C02766=1037.489,91.747,407.519,169.496,40.208,157.561
C02767=1037.483,91.497,407.538,169.494,40.208,157.561
C02768=1037.477,91.248,407.557,169.492,40.208,157.561
C02769=1037.471,90.999,407.575,169.490,40.208,157.561
C02770=1037.465,90.749,407.595,169.488,40.208,157.561
C02771=1037.458,90.500,407.613,169.486,40.208,157.561
C02772=1037.452,90.252,407.633,169.484,40.208,157.561
C02773=1037.446,90.002,407.652,169.482,40.208,157.561
C02774=1037.440,89.753,407.671,169.480,40.207,157.561
C02775=1037.434,89.504,407.690,169.478,40.207,157.560
C02776=1037.427,89.254,407.709,169.476,40.208,157.560
C02777=1037.420,89.005,407.728,169.473,40.207,157.560
C02778=1037.414,88.756,407.746,169.471,40.207,157.560
C02779=1037.408,88.506,407.765,169.469,40.208,157.560
C02780=1037.402,88.257,407.784,169.467,40.208,157.560
C02781=1037.396,88.008,407.803,169.465,40.207,157.560
C02782=1037.389,87.759,407.821,169.463,40.208,157.560
C02783=1037.383,87.510,407.840,169.461,40.208,157.560
C02784=1037.377,87.260,407.859,169.459,40.207,157.560
C02785=1037.371,87.011,407.878,169.457,40.208,157.560
C02786=1037.364,86.762,407.897,169.455,40.208,157.560
C02787=1037.358,86.513,407.915,169.453,40.207,157.559
C02788=1037.351,86.264,407.934,169.451,40.207,157.559
C02789=1037.346,86.014,407.953,169.449,40.208,157.559
C02790=1037.339,85.765,407.972,169.447,40.207,157.559
C02791=1037.333,85.516,407.990,169.444,40.207,157.559
C02792=1037.326,85.267,408.009,169.442,40.208,157.559
C02793=1037.320,85.018,408.028,169.439,40.207,157.559
C02794=1037.314,84.769,408.047,169.437,40.207,157.559
C02795=1037.308,84.519,408.066,169.435,40.208,157.559
C02796=1037.301,84.270,408.084,169.433,40.207,157.559
C02797=1037.295,84.021,408.103,169.431,40.207,157.559
C02798=1037.289,83.771,408.121,169.429,40.208,157.558
C02799=1037.283,83.522,408.140,169.427,40.207,157.558
C02800=1037.277,83.273,408.159,169.425,40.207,157.558
C02801=1037.270,83.024,408.177,169.423,40.208,157.558
C02802=1037.264,82.775,408.196,169.421,40.207,157.558
C02803=1037.257,82.526,408.215,169.419,40.207,157.558
C02804=1037.251,82.276,408.233,169.417,40.207,157.558
C02805=1037.245,82.027,408.253,169.415,40.207,157.558
C02806=1037.239,81.777,408.270,169.413,40.207,157.558
C02807=1037.233,81.528,408.289,169.410,40.207,157.558
C02808=1037.226,81.279,408.308,169.408,40.207,157.557
C02809=1037.220,81.031,408.326,169.406,40.207,157.557
C02810=1037.214,80.781,408.345,169.404,40.207,157.557
C02811=1037.208,80.532,408.364,169.402,40.207,157.557
C02812=1037.202,80.282,408.382,169.400,40.207,157.557
C02813=1037.196,80.033,408.401,169.398,40.207,157.557
C02814=1037.189,79.784,408.419,169.396,40.207,157.557
C02815=1037.183,79.535,408.438,169.394,40.206,157.557
C02816=1037.177,79.285,408.456,169.392,40.207,157.557
C02817=1037.171,79.036,408.475,169.390,40.207,157.557
C02818=1037.165,78.787,408.494,169.388,40.206,157.556
C02819=1037.159,78.538,408.512,169.386,40.206,157.556
C02820=1037.153,78.288,408.530,169.383,40.206,157.556
C02821=1037.146,78.039,408.549,169.381,40.206,157.556
C02822=1037.140,77.790,408.567,169.379,40.206,157.556
C02823=1037.134,77.541,408.586,169.377,40.207,157.556
C02824=1037.127,77.291,408.604,169.375,40.206,157.556
C02825=1037.118,76.901,408.633,169.372,40.206,157.556
C02826=1037.108,76.512,408.661,169.369,40.206,157.556
C02827=1037.098,76.122,408.690,169.365,40.207,157.556
C02828=1037.088,75.733,408.718,169.362,40.206,157.555
C02829=1037.081,75.484,408.737,169.360,40.206,157.555
C02830=1037.076,75.235,408.755,169.358,40.207,157.555
C02831=1037.070,74.985,408.773,169.356,40.207,157.555
C02832=1037.063,74.736,408.792,169.353,40.206,157.555
C02833=1037.057,74.487,408.810,169.351,40.206,157.555
C02834=1037.051,74.237,408.828,169.349,40.207,157.555
C02835=1037.044,73.988,408.846,169.347,40.207,157.555
C02836=1037.037,73.739,408.864,169.345,40.206,157.555
C02837=1037.032,73.490,408.882,169.343,40.207,157.555
C02838=1037.025,73.241,408.900,169.341,40.207,157.555
C02839=1037.019,72.992,408.919,169.339,40.206,157.554
C02840=1037.013,72.742,408.937,169.337,40.207,157.554
C02841=1037.006,72.493,408.956,169.335,40.207,157.554
C02842=1037.001,72.244,408.973,169.333,40.206,157.554
C02843=1036.994,71.995,408.992,169.331,40.206,157.554
C02844=1036.988,71.745,409.010,169.329,40.207,157.554
C02845=1036.981,71.496,409.028,169.327,40.207,157.554
C02846=1036.975,71.246,409.046,169.325,40.206,157.554
C02847=1036.969,70.997,409.064,169.323,40.207,157.554
C02848=1036.963,70.748,409.082,169.321,40.207,157.554
C02849=1036.957,70.498,409.100,169.318,40.206,157.554
C02850=1036.951,70.249,409.119,169.316,40.207,157.554
C02851=1036.944,70.000,409.136,169.314,40.207,157.553
C02852=1036.938,69.751,409.154,169.312,40.207,157.553
C02853=1036.932,69.502,409.172,169.310,40.206,157.553
C02854=1036.926,69.252,409.190,169.308,40.207,157.553
C02855=1036.919,69.003,409.209,169.305,40.207,157.553
C02856=1036.912,68.753,409.226,169.303,40.207,157.553
C02857=1036.906,68.505,409.244,169.301,40.207,157.553
C02858=1036.900,68.255,409.262,169.299,40.207,157.553
C02859=1036.894,68.005,409.280,169.297,40.207,157.553
C02860=1036.887,67.757,409.298,169.295,40.207,157.553
C02861=1036.882,67.508,409.316,169.293,40.207,157.553
C02862=1036.875,67.258,409.334,169.291,40.207,157.553
C02863=1036.868,67.009,409.352,169.289,40.207,157.553
C02864=1036.862,66.759,409.370,169.286,40.207,157.552
C02865=1036.857,66.510,409.387,169.284,40.207,157.552
C02866=1036.850,66.261,409.406,169.282,40.207,157.552
C02867=1036.843,66.012,409.423,169.280,40.207,157.552
C02868=1036.837,65.762,409.441,169.278,40.208,157.552
C02869=1036.831,65.513,409.458,169.276,40.207,157.552
C02870=1036.825,65.264,409.477,169.274,40.207,157.552
C02871=1036.818,65.014,409.495,169.272,40.208,157.552
C02872=1036.812,64.765,409.512,169.270,40.208,157.552
C02873=1036.806,64.516,409.530,169.268,40.207,157.552
C02874=1036.800,64.267,409.548,169.266,40.207,157.552
C02875=1036.793,64.017,409.566,169.264,40.208,157.552
C02876=1036.787,63.768,409.583,169.262,40.208,157.551
C02877=1036.777,63.373,409.611,169.258,40.208,157.551
C02878=1036.767,62.978,409.638,169.255,40.208,157.551
C02879=1036.756,62.583,409.667,169.252,40.208,157.551
C02880=1036.746,62.188,409.695,169.249,40.208,157.551
C02881=1036.739,61.939,409.712,169.246,40.209,157.551
C02882=1036.733,61.689,409.730,169.244,40.209,157.551
C02883=1036.727,61.440,409.747,169.242,40.209,157.551
C02884=1036.720,61.191,409.764,169.240,40.209,157.551
C02885=1036.713,60.904,409.785,169.237,40.209,157.551
C02886=1036.706,60.618,409.805,169.234,40.209,157.551
C02887=1036.698,60.332,409.825,169.232,40.209,157.551
C02888=1036.691,60.046,409.845,169.230,40.210,157.550
C02889=1036.684,59.796,409.862,169.228,40.210,157.550
C02890=1036.679,59.547,409.880,169.226,40.210,157.550
C02891=1036.672,59.298,409.897,169.223,40.210,157.550
C02892=1036.665,59.049,409.915,169.221,40.210,157.550
C02893=1036.660,58.800,409.932,169.219,40.210,157.550
C02894=1036.653,58.550,409.949,169.217,40.210,157.550
C02895=1036.646,58.301,409.967,169.215,40.210,157.550
C02896=1036.640,58.052,409.984,169.213,40.211,157.550
C02897=1036.633,57.802,410.002,169.211,40.211,157.550
C02898=1036.627,57.553,410.019,169.209,40.211,157.550
C02899=1036.621,57.304,410.037,169.207,40.211,157.550
C02900=1036.614,57.054,410.054,169.205,40.211,157.550
C02901=1036.608,56.805,410.072,169.203,40.211,157.550
C02902=1036.602,56.556,410.089,169.201,40.211,157.550
C02903=1036.595,56.306,410.106,169.199,40.211,157.549
C02904=1036.589,56.057,410.124,169.197,40.211,157.549
C02905=1036.583,55.808,410.141,169.194,40.212,157.549
C02906=1036.576,55.558,410.158,169.192,40.212,157.549
C02907=1036.570,55.309,410.176,169.189,40.211,157.549
C02908=1036.563,55.060,410.193,169.187,40.212,157.549
C02909=1036.557,54.811,410.210,169.185,40.212,157.549
C02910=1036.551,54.561,410.228,169.183,40.212,157.549
C02911=1036.544,54.311,410.245,169.181,40.212,157.549
C02912=1036.538,54.063,410.262,169.179,40.212,157.549
C02913=1036.532,53.813,410.280,169.177,40.212,157.549
C02914=1036.526,53.564,410.297,169.175,40.212,157.549
C02915=1036.519,53.315,410.314,169.173,40.212,157.549
C02916=1036.513,53.066,410.332,169.171,40.213,157.549
C02917=1036.507,52.816,410.348,169.169,40.213,157.549
C02918=1036.500,52.566,410.366,169.167,40.212,157.548
C02919=1036.495,52.317,410.383,169.165,40.213,157.548
C02920=1036.488,52.068,410.401,169.163,40.213,157.548
C02921=1036.481,51.819,410.418,169.161,40.213,157.548
C02922=1036.476,51.569,410.435,169.158,40.213,157.548
C02923=1036.469,51.320,410.452,169.156,40.213,157.548
C02924=1036.462,51.071,410.469,169.154,40.213,157.548
C02925=1036.457,50.822,410.487,169.152,40.213,157.548
C02926=1036.450,50.572,410.504,169.150,40.213,157.548
C02927=1036.444,50.323,410.520,169.148,40.214,157.548
C02928=1036.437,50.073,410.538,169.145,40.213,157.548
C02929=1036.432,49.824,410.555,169.143,40.213,157.548
C02930=1036.425,49.575,410.572,169.141,40.213,157.547
C02931=1036.419,49.326,410.589,169.139,40.214,157.547
C02932=1036.413,49.076,410.607,169.137,40.214,157.547
C02933=1036.407,48.827,410.624,169.135,40.213,157.547
C02934=1036.400,48.578,410.641,169.133,40.214,157.547
C02935=1036.395,48.328,410.658,169.131,40.214,157.547
C02936=1036.388,48.079,410.675,169.129,40.214,157.547
C02937=1036.381,47.830,410.692,169.127,40.214,157.547
C02938=1036.375,47.580,410.709,169.125,40.214,157.547
C02939=1036.369,47.331,410.726,169.123,40.214,157.547
C02940=1036.362,47.081,410.744,169.120,40.214,157.547
C02941=1036.357,46.832,410.760,169.118,40.214,157.547
C02942=1036.351,46.583,410.777,169.116,40.214,157.546
C02943=1036.344,46.333,410.795,169.114,40.214,157.546
C02944=1036.338,46.084,410.811,169.112,40.214,157.546
C02945=1036.332,45.834,410.829,169.110,40.215,157.546
C02946=1036.326,45.586,410.846,169.107,40.214,157.546
C02947=1036.320,45.336,410.862,169.105,40.214,157.546
C02948=1036.313,45.087,410.880,169.103,40.214,157.546
C02949=1036.306,44.800,410.899,169.101,40.215,157.546
C02950=1036.299,44.514,410.919,169.098,40.214,157.546
C02951=1036.292,44.227,410.938,169.096,40.214,157.546
C02952=1036.285,43.941,410.958,169.094,40.215,157.546
C02953=1036.279,43.691,410.975,169.092,40.214,157.546
C02954=1036.273,43.442,410.991,169.090,40.214,157.545
C02955=1036.267,43.193,411.009,169.088,40.215,157.545
C02956=1036.261,42.943,411.025,169.085,40.215,157.545
C02957=1036.254,42.694,411.042,169.083,40.215,157.545
C02958=1036.248,42.444,411.059,169.081,40.215,157.545
C02959=1036.242,42.195,411.076,169.079,40.215,157.545
C02960=1036.236,41.946,411.092,169.077,40.215,157.545
C02961=1036.229,41.696,411.110,169.075,40.215,157.545
C02962=1036.223,41.447,411.126,169.073,40.215,157.545
C02963=1036.216,41.198,411.143,169.071,40.216,157.545
C02964=1036.210,40.948,411.159,169.069,40.216,157.545
C02965=1036.204,40.700,411.176,169.067,40.216,157.545
C02966=1036.197,40.450,411.193,169.065,40.216,157.545
C02967=1036.191,40.200,411.209,169.061,40.216,157.545
C02968=1036.185,39.951,411.226,169.059,40.216,157.544
C02969=1036.178,39.701,411.243,169.057,40.216,157.544
C02970=1036.172,39.453,411.260,169.055,40.216,157.544
C02971=1036.166,39.203,411.276,169.053,40.217,157.544
C02972=1036.160,38.953,411.293,169.051,40.217,157.544
C02973=1036.153,38.705,411.310,169.049,40.217,157.544
C02974=1036.147,38.454,411.326,169.047,40.217,157.544
C02975=1036.141,38.205,411.343,169.045,40.217,157.544
C02976=1036.135,37.956,411.359,169.043,40.217,157.544
C02977=1036.128,37.706,411.376,169.041,40.217,157.544
C02978=1036.122,37.457,411.392,169.038,40.217,157.544
C02979=1036.116,37.208,411.409,169.036,40.218,157.544
C02980=1036.109,36.958,411.426,169.034,40.218,157.544
C02981=1036.103,36.709,411.442,169.032,40.218,157.544
C02982=1036.097,36.460,411.458,169.030,40.218,157.544
C02983=1036.090,36.210,411.475,169.028,40.218,157.543
C02984=1036.084,35.961,411.491,169.026,40.218,157.543
C02985=1036.078,35.712,411.508,169.024,40.218,157.543
C02986=1036.071,35.462,411.524,169.021,40.218,157.543
C02987=1036.065,35.213,411.540,169.019,40.219,157.543
C02988=1036.058,34.964,411.557,169.017,40.219,157.543
C02989=1036.052,34.714,411.574,169.015,40.219,157.543
C02990=1036.046,34.465,411.590,169.013,40.219,157.543
C02991=1036.039,34.215,411.606,169.011,40.219,157.543
C02992=1036.033,33.965,411.622,169.009,40.220,157.543
C02993=1036.026,33.717,411.639,169.006,40.220,157.543
C02994=1036.020,33.467,411.655,169.003,40.220,157.543
C02995=1036.014,33.218,411.671,169.001,40.220,157.543
C02996=1036.007,32.968,411.688,168.999,40.220,157.543
C02997=1036.001,32.719,411.704,168.997,40.221,157.543
C02998=1035.995,32.470,411.720,168.995,40.221,157.543
C02999=1035.989,32.219,411.737,168.993,40.221,157.543
C03000=1035.982,31.971,411.753,168.991,40.221,157.543
C03001=1035.976,31.722,411.769,168.989,40.221,157.543
C03002=1035.970,31.472,411.786,168.986,40.221,157.542
C03003=1035.963,31.222,411.802,168.984,40.221,157.542
C03004=1035.957,30.973,411.818,168.982,40.221,157.542
C03005=1035.951,30.724,411.834,168.980,40.222,157.542
C03006=1035.945,30.475,411.850,168.978,40.222,157.542
C03007=1035.939,30.225,411.867,168.976,40.222,157.542
C03008=1035.931,29.976,411.883,168.974,40.222,157.542
C03009=1035.926,29.726,411.899,168.971,40.222,157.542
C03010=1035.920,29.477,411.915,168.969,40.223,157.542
C03011=1035.914,29.227,411.932,168.967,40.223,157.542
C03012=1035.906,28.978,411.948,168.965,40.223,157.542
C03013=1035.900,28.691,411.967,168.963,40.223,157.542
C03014=1035.892,28.405,411.985,168.960,40.223,157.542
C03015=1035.885,28.119,412.004,168.958,40.223,157.542
C03016=1035.878,27.832,412.022,168.955,40.223,157.541
C03017=1035.872,27.582,412.038,168.953,40.224,157.541
C03018=1035.865,27.333,412.054,168.951,40.224,157.541
C03019=1035.859,27.083,412.071,168.949,40.224,157.541
C03020=1035.852,26.834,412.086,168.947,40.224,157.541
C03021=1035.846,26.585,412.102,168.945,40.224,157.541
C03022=1035.839,26.336,412.118,168.941,40.225,157.541
C03023=1035.833,26.087,412.134,168.939,40.225,157.541
C03024=1035.827,25.837,412.151,168.937,40.225,157.541
C03025=1035.820,25.587,412.166,168.935,40.225,157.541
C03026=1035.814,25.338,412.182,168.933,40.225,157.541
C03027=1035.808,25.089,412.198,168.931,40.226,157.541
C03028=1035.802,24.839,412.214,168.928,40.226,157.541
C03029=1035.795,24.590,412.230,168.926,40.226,157.541
C03030=1035.789,24.340,412.246,168.924,40.226,157.541
C03031=1035.782,24.091,412.262,168.922,40.226,157.541
C03032=1035.776,23.841,412.278,168.920,40.227,157.541
C03033=1035.770,23.592,412.293,168.918,40.227,157.541
C03034=1035.764,23.343,412.310,168.915,40.227,157.540
C03035=1035.757,23.094,412.325,168.913,40.227,157.540
C03036=1035.751,22.844,412.341,168.911,40.228,157.540
C03037=1035.744,22.594,412.357,168.909,40.228,157.540
C03038=1035.738,22.345,412.373,168.907,40.228,157.540
C03039=1035.731,22.096,412.389,168.904,40.228,157.540
C03040=1035.725,21.846,412.405,168.902,40.228,157.540
C03041=1035.719,21.597,412.420,168.900,40.229,157.540
C03042=1035.713,21.347,412.436,168.898,40.229,157.540
C03043=1035.706,21.098,412.452,168.896,40.229,157.540
C03044=1035.700,20.849,412.468,168.894,40.229,157.540
C03045=1035.694,20.599,412.483,168.891,40.229,157.540
C03046=1035.687,20.349,412.500,168.889,40.230,157.540
C03047=1035.681,20.100,412.515,168.887,40.230,157.540
C03048=1035.675,19.851,412.532,168.885,40.230,157.540
C03049=1035.668,19.601,412.547,168.883,40.230,157.540
C03050=1035.662,19.352,412.563,168.881,40.230,157.540
C03051=1035.656,19.103,412.578,168.878,40.231,157.540
C03052=1035.649,18.853,412.593,168.876,40.231,157.540
C03053=1035.643,18.604,412.610,168.874,40.231,157.539
C03054=1035.637,18.354,412.625,168.872,40.231,157.539
C03055=1035.630,18.105,412.640,168.870,40.232,157.539
C03056=1035.624,17.856,412.656,168.867,40.232,157.539
C03057=1035.618,17.606,412.671,168.865,40.233,157.539
C03058=1035.611,17.357,412.687,168.863,40.233,157.539
C03059=1035.606,17.107,412.703,168.861,40.233,157.539
C03060=1035.598,16.857,412.719,168.859,40.233,157.539
C03061=1035.592,16.608,412.735,168.856,40.234,157.539
C03062=1035.586,16.358,412.750,168.854,40.234,157.539
C03063=1035.579,16.109,412.766,168.852,40.234,157.539
C03064=1035.574,15.859,412.781,168.850,40.234,157.539
C03065=1035.567,15.610,412.797,168.848,40.234,157.539
C03066=1035.561,15.361,412.812,168.845,40.235,157.539
C03067=1035.555,15.111,412.828,168.843,40.235,157.539
C03068=1035.548,14.862,412.844,168.841,40.235,157.539
C03069=1035.542,14.612,412.859,168.838,40.235,157.539
C03070=1035.536,14.363,412.874,168.836,40.235,157.539
C03071=1035.529,14.113,412.890,168.833,40.236,157.539
C03072=1035.523,13.864,412.905,168.831,40.236,157.539
C03073=1035.516,13.615,412.920,168.829,40.236,157.538
C03074=1035.510,13.365,412.935,168.827,40.236,157.538
C03075=1035.504,13.116,412.952,168.824,40.237,157.538
C03076=1035.498,12.866,412.967,168.822,40.237,157.538
C03077=1035.490,12.581,412.984,168.820,40.238,157.538
C03078=1035.482,12.296,413.002,168.817,40.238,157.538
C03079=1035.475,12.010,413.019,168.814,40.238,157.538
C03080=1035.468,11.725,413.036,168.812,40.238,157.538
C03081=1035.462,11.476,413.051,168.810,40.239,157.538
C03082=1035.455,11.227,413.067,168.807,40.239,157.538
C03083=1035.449,10.977,413.082,168.805,40.240,157.538
C03084=1035.442,10.728,413.097,168.803,40.240,157.538
C03085=1035.436,10.478,413.112,168.801,40.240,157.538
C03086=1035.429,10.229,413.127,168.798,40.240,157.538
C03087=1035.423,9.979,413.142,168.796,40.241,157.538
C03088=1035.416,9.730,413.158,168.794,40.241,157.538
C03089=1035.410,9.480,413.173,168.792,40.242,157.538
C03090=1035.404,9.231,413.188,168.789,40.242,157.538
C03091=1035.398,8.981,413.204,168.787,40.242,157.538
C03092=1035.391,8.732,413.219,168.785,40.242,157.538
C03093=1035.385,8.482,413.234,168.783,40.242,157.538
C03094=1035.378,8.233,413.250,168.780,40.243,157.538
C03095=1035.372,7.983,413.265,168.778,40.244,157.538
C03096=1035.365,7.734,413.279,168.776,40.244,157.538
C03097=1035.359,7.484,413.294,168.774,40.244,157.538
C03098=1035.353,7.234,413.309,168.771,40.244,157.538
C03099=1035.347,6.986,413.325,168.769,40.244,157.537
C03100=1035.340,6.736,413.340,168.767,40.245,157.537
C03101=1035.334,6.487,413.355,168.764,40.245,157.537
C03102=1035.327,6.237,413.369,168.762,40.246,157.537
C03103=1035.321,5.988,413.385,168.760,40.246,157.537
C03104=1035.314,5.738,413.400,168.758,40.246,157.537
C03105=1035.308,5.489,413.415,168.755,40.246,157.537
C03106=1035.302,5.239,413.430,168.753,40.247,157.537
C03107=1035.296,4.990,413.445,168.751,40.247,157.537
C03108=1035.289,4.740,413.460,168.749,40.247,157.537
C03109=1035.283,4.491,413.475,168.746,40.247,157.537
C03110=1035.276,4.242,413.490,168.744,40.248,157.537
C03111=1035.270,3.992,413.505,168.742,40.248,157.537
C03112=1035.264,3.742,413.521,168.740,40.249,157.537
C03113=1035.258,3.492,413.536,168.737,40.249,157.537
C03114=1035.252,3.243,413.550,168.735,40.249,157.537
C03115=1035.246,2.994,413.565,168.733,40.249,157.537
C03116=1035.239,2.744,413.580,168.731,40.249,157.537
C03117=1035.233,2.495,413.596,168.728,40.250,157.537
C03118=1035.226,2.245,413.611,168.726,40.250,157.537
C03119=1035.220,1.996,413.625,168.724,40.250,157.537
C03120=1035.214,1.747,413.640,168.721,40.251,157.537
C03121=1035.208,1.497,413.655,168.719,40.251,157.537
C03122=1035.201,1.248,413.670,168.717,40.251,157.537
C03123=1035.195,0.998,413.685,168.715,40.252,157.536
C03124=1035.189,0.749,413.700,168.712,40.252,157.536
C03125=1035.183,0.499,413.715,168.710,40.252,157.536
C03126=1035.176,0.250,413.729,168.708,40.252,157.536
C03127=1035.170,-0.000,413.744,168.706,40.253,157.536
C03128=1035.164,-0.249,413.759,168.703,40.253,157.536
C03129=1035.158,-0.499,413.774,168.701,40.253,157.536
C03130=1035.151,-0.748,413.789,168.699,40.253,157.536
C03131=1035.145,-0.998,413.804,168.696,40.254,157.536
C03132=1035.139,-1.247,413.818,168.694,40.254,157.536
C03133=1035.133,-1.497,413.833,168.692,40.255,157.536
C03134=1035.127,-1.746,413.848,168.690,40.255,157.536
C03135=1035.120,-1.996,413.863,168.687,40.255,157.536
C03136=1035.114,-2.245,413.878,168.685,40.255,157.536
C03137=1035.108,-2.495,413.893,168.683,40.255,157.536
C03138=1035.102,-2.744,413.908,168.680,40.256,157.536
C03139=1035.096,-2.993,413.922,168.678,40.256,157.536
C03140=1035.089,-3.243,413.937,168.676,40.256,157.536
C03141=1035.082,-3.526,413.954,168.673,40.256,157.536
C03142=1035.075,-3.810,413.970,168.671,40.257,157.536
C03143=1035.068,-4.093,413.986,168.668,40.258,157.536
C03144=1035.060,-4.377,414.004,168.665,40.258,157.535
C03145=1035.055,-4.626,414.018,168.663,40.258,157.535
C03146=1035.048,-4.876,414.032,168.661,40.259,157.535
C03147=1035.041,-5.125,414.047,168.658,40.259,157.535
C03148=1035.035,-5.374,414.061,168.656,40.259,157.535
C03149=1035.028,-5.624,414.076,168.654,40.260,157.535
C03150=1035.022,-5.874,414.090,168.651,40.261,157.535
C03151=1035.016,-6.124,414.105,168.649,40.261,157.535
C03152=1035.009,-6.372,414.119,168.647,40.261,157.535
C03153=1035.003,-6.622,414.134,168.644,40.261,157.535
C03154=1034.997,-6.872,414.148,168.642,40.262,157.535
C03155=1034.990,-7.121,414.162,168.640,40.262,157.535
C03156=1034.984,-7.370,414.177,168.637,40.263,157.535
C03157=1034.978,-7.621,414.191,168.635,40.263,157.535
C03158=1034.971,-7.869,414.205,168.632,40.264,157.535
C03159=1034.965,-8.119,414.220,168.630,40.264,157.535
C03160=1034.959,-8.369,414.234,168.628,40.264,157.535
C03161=1034.952,-8.618,414.248,168.625,40.264,157.535
C03162=1034.946,-8.868,414.263,168.623,40.265,157.535
C03163=1034.940,-9.118,414.278,168.621,40.265,157.535
C03164=1034.933,-9.367,414.292,168.618,40.266,157.535
C03165=1034.927,-9.616,414.307,168.616,40.266,157.535
C03166=1034.921,-9.866,414.321,168.614,40.267,157.535
C03167=1034.914,-10.115,414.335,168.611,40.267,157.535
C03168=1034.908,-10.365,414.350,168.609,40.267,157.535
C03169=1034.902,-10.614,414.363,168.607,40.267,157.535
C03170=1034.895,-10.864,414.378,168.604,40.268,157.535
C03171=1034.889,-11.114,414.392,168.602,40.269,157.535
C03172=1034.883,-11.363,414.406,168.599,40.269,157.535
C03173=1034.876,-11.612,414.421,168.597,40.269,157.535
C03174=1034.871,-11.862,414.435,168.595,40.270,157.535
C03175=1034.864,-12.111,414.449,168.592,40.270,157.535
C03176=1034.858,-12.361,414.464,168.590,40.270,157.535
C03177=1034.851,-12.610,414.478,168.588,40.271,157.535
C03178=1034.845,-12.860,414.492,168.585,40.272,157.535
C03179=1034.839,-13.109,414.506,168.583,40.272,157.535
C03180=1034.833,-13.359,414.520,168.581,40.272,157.534
C03181=1034.827,-13.608,414.535,168.578,40.272,157.534
C03182=1034.821,-13.859,414.549,168.576,40.272,157.534
C03183=1034.814,-14.107,414.563,168.573,40.273,157.534
C03184=1034.808,-14.357,414.577,168.571,40.274,157.534
C03185=1034.802,-14.606,414.591,168.569,40.274,157.534
C03186=1034.796,-14.856,414.605,168.566,40.274,157.534
C03187=1034.789,-15.106,414.620,168.564,40.275,157.534
C03188=1034.783,-15.355,414.633,168.562,40.275,157.534
C03189=1034.777,-15.605,414.648,168.559,40.275,157.534
C03190=1034.770,-15.854,414.662,168.557,40.276,157.534
C03191=1034.763,-16.104,414.676,168.554,40.277,157.534
C03192=1034.758,-16.353,414.690,168.552,40.277,157.534
C03193=1034.751,-16.603,414.704,168.549,40.278,157.534
C03194=1034.745,-16.852,414.718,168.547,40.278,157.534
C03195=1034.738,-17.102,414.732,168.545,40.278,157.534
C03196=1034.732,-17.351,414.745,168.542,40.279,157.534
C03197=1034.726,-17.601,414.760,168.540,40.279,157.534
C03198=1034.720,-17.850,414.773,168.537,40.280,157.534
C03199=1034.713,-18.100,414.787,168.535,40.280,157.534
C03200=1034.707,-18.349,414.801,168.532,40.281,157.534
C03201=1034.700,-18.599,414.815,168.531,40.282,157.534
C03202=1034.694,-18.848,414.828,168.529,40.282,157.534
C03203=1034.688,-19.098,414.843,168.525,40.282,157.534
C03204=1034.681,-19.347,414.857,168.524,40.283,157.534
C03205=1034.674,-19.630,414.872,168.521,40.283,157.534
C03206=1034.667,-19.911,414.888,168.518,40.283,157.534
C03207=1034.660,-20.193,414.904,168.516,40.284,157.534
C03208=1034.653,-20.474,414.919,168.513,40.285,157.534
C03209=1034.646,-20.724,414.932,168.510,40.286,157.534
C03210=1034.640,-20.973,414.947,168.508,40.286,157.534
C03211=1034.634,-21.223,414.961,168.505,40.286,157.534
C03212=1034.627,-21.473,414.974,168.503,40.287,157.534
C03213=1034.621,-21.723,414.988,168.501,40.287,157.534
C03214=1034.615,-21.972,415.001,168.498,40.287,157.534
C03215=1034.608,-22.221,415.016,168.496,40.288,157.534
C03216=1034.603,-22.471,415.030,168.493,40.289,157.534
C03217=1034.596,-22.720,415.043,168.491,40.289,157.534
C03218=1034.589,-22.970,415.057,168.488,40.290,157.534
C03219=1034.584,-23.220,415.070,168.486,40.290,157.534
C03220=1034.577,-23.470,415.084,168.483,40.290,157.534
C03221=1034.571,-23.718,415.098,168.481,40.291,157.534
C03222=1034.565,-23.968,415.112,168.479,40.291,157.534
C03223=1034.558,-24.218,415.126,168.476,40.291,157.533
C03224=1034.552,-24.467,415.139,168.474,40.292,157.534
C03225=1034.547,-24.717,415.153,168.471,40.293,157.533
C03226=1034.540,-24.967,415.166,168.469,40.293,157.534
C03227=1034.534,-25.216,415.180,168.466,40.294,157.533
C03228=1034.528,-25.466,415.193,168.464,40.294,157.533
C03229=1034.521,-25.716,415.207,168.461,40.295,157.533
C03230=1034.515,-25.965,415.220,168.459,40.295,157.533
C03231=1034.510,-26.214,415.234,168.457,40.295,157.533
C03232=1034.503,-26.464,415.249,168.454,40.296,157.533
C03233=1034.496,-26.713,415.262,168.452,40.296,157.533
C03234=1034.490,-26.963,415.275,168.449,40.297,157.533
C03235=1034.484,-27.213,415.289,168.447,40.298,157.533
C03236=1034.478,-27.462,415.303,168.444,40.298,157.533
C03237=1034.471,-27.712,415.316,168.442,40.299,157.533
C03238=1034.465,-27.962,415.329,168.439,40.299,157.533
C03239=1034.459,-28.211,415.342,168.437,40.300,157.533
C03240=1034.452,-28.461,415.356,168.434,40.300,157.533
C03241=1034.446,-28.710,415.369,168.433,40.301,157.533
C03242=1034.440,-28.959,415.382,168.429,40.301,157.533
C03243=1034.433,-29.209,415.396,168.428,40.302,157.533
C03244=1034.427,-29.459,415.409,168.425,40.303,157.533
C03245=1034.420,-29.708,415.422,168.423,40.303,157.533
C03246=1034.414,-29.957,415.436,168.420,40.304,157.533
C03247=1034.407,-30.207,415.449,168.418,40.305,157.533
C03248=1034.401,-30.457,415.462,168.415,40.305,157.533
C03249=1034.395,-30.706,415.475,168.413,40.305,157.533
C03250=1034.389,-30.957,415.489,168.410,40.306,157.533
C03251=1034.383,-31.206,415.503,168.408,40.306,157.533
C03252=1034.377,-31.455,415.516,168.405,40.307,157.533
C03253=1034.371,-31.704,415.529,168.403,40.307,157.533
C03254=1034.364,-31.955,415.542,168.400,40.308,157.533
C03255=1034.358,-32.204,415.555,168.398,40.308,157.533
C03256=1034.352,-32.453,415.569,168.395,40.309,157.533
C03257=1034.345,-32.703,415.582,168.392,40.310,157.533
C03258=1034.339,-32.953,415.596,168.390,40.311,157.533
C03259=1034.333,-33.203,415.608,168.387,40.311,157.533
C03260=1034.326,-33.452,415.621,168.385,40.312,157.533
C03261=1034.320,-33.701,415.635,168.382,40.312,157.533
C03262=1034.313,-33.951,415.648,168.380,40.313,157.533
C03263=1034.308,-34.201,415.661,168.377,40.313,157.533
C03264=1034.301,-34.450,415.674,168.375,40.314,157.533
C03265=1034.295,-34.700,415.687,168.372,40.314,157.533
C03266=1034.289,-34.949,415.701,168.370,40.315,157.533
C03267=1034.282,-35.199,415.714,168.367,40.315,157.533
C03268=1034.276,-35.449,415.727,168.366,40.316,157.533
C03269=1034.269,-35.729,415.741,168.363,40.317,157.533
C03270=1034.262,-36.010,415.757,168.360,40.318,157.533
C03271=1034.255,-36.292,415.771,168.357,40.318,157.533
C03272=1034.248,-36.572,415.786,168.354,40.319,157.533
C03273=1034.242,-36.822,415.798,168.352,40.319,157.533
C03274=1034.235,-37.072,415.812,168.349,40.320,157.533
C03275=1034.229,-37.321,415.825,168.347,40.320,157.533
C03276=1034.223,-37.571,415.838,168.344,40.321,157.533
C03277=1034.217,-37.820,415.851,168.342,40.321,157.533
C03278=1034.211,-38.070,415.864,168.339,40.322,157.533
C03279=1034.205,-38.319,415.877,168.337,40.322,157.533
C03280=1034.199,-38.569,415.890,168.334,40.323,157.533
C03281=1034.193,-38.819,415.903,168.332,40.324,157.533
C03282=1034.186,-39.068,415.916,168.329,40.325,157.533
C03283=1034.180,-39.318,415.929,168.326,40.325,157.533
C03284=1034.174,-39.568,415.942,168.324,40.326,157.533
C03285=1034.167,-39.817,415.954,168.321,40.327,157.533
C03286=1034.161,-40.066,415.967,168.319,40.327,157.533
C03287=1034.155,-40.316,415.980,168.316,40.328,157.533
C03288=1034.149,-40.566,415.993,168.313,40.328,157.533
C03289=1034.142,-40.815,416.005,168.311,40.329,157.533
C03290=1034.135,-41.065,416.019,168.309,40.330,157.533
C03291=1034.129,-41.315,416.031,168.307,40.330,157.533
C03292=1034.123,-41.564,416.045,168.304,40.331,157.533
C03293=1034.117,-41.814,416.057,168.301,40.332,157.533
C03294=1034.111,-42.064,416.069,168.299,40.332,157.533
C03295=1034.104,-42.313,416.082,168.296,40.333,157.533
C03296=1034.099,-42.563,416.095,168.294,40.333,157.533
C03297=1034.092,-42.812,416.108,168.291,40.334,157.533
C03298=1034.086,-43.062,416.120,168.288,40.335,157.533
C03299=1034.079,-43.311,416.134,168.286,40.336,157.533
C03300=1034.074,-43.561,416.146,168.283,40.336,157.533
C03301=1034.067,-43.810,416.158,168.281,40.337,157.533
C03302=1034.061,-44.060,416.171,168.278,40.338,157.533
C03303=1034.055,-44.310,416.184,168.275,40.339,157.533
C03304=1034.048,-44.560,416.196,168.273,40.339,157.533
C03305=1034.041,-44.809,416.209,168.270,40.340,157.533
C03306=1034.035,-45.059,416.222,168.269,40.341,157.533
C03307=1034.030,-45.309,416.235,168.265,40.341,157.533
C03308=1034.023,-45.558,416.247,168.263,40.342,157.533
C03309=1034.017,-45.808,416.260,168.261,40.343,157.533
C03310=1034.011,-46.058,416.272,168.258,40.343,157.533
C03311=1034.004,-46.307,416.285,168.256,40.344,157.533
C03312=1033.998,-46.556,416.298,168.253,40.344,157.533
C03313=1033.992,-46.806,416.310,168.250,40.345,157.533
C03314=1033.987,-47.056,416.322,168.248,40.346,157.533
C03315=1033.980,-47.304,416.335,168.245,40.346,157.533
C03316=1033.974,-47.554,416.348,168.243,40.347,157.533
C03317=1033.968,-47.804,416.360,168.240,40.348,157.533
C03318=1033.961,-48.054,416.372,168.237,40.348,157.533
C03319=1033.955,-48.303,416.385,168.235,40.349,157.533
C03320=1033.949,-48.553,416.398,168.232,40.350,157.533
C03321=1033.942,-48.803,416.410,168.229,40.351,157.533
C03322=1033.937,-49.052,416.422,168.227,40.351,157.533
C03323=1033.931,-49.302,416.435,168.224,40.352,157.533
C03324=1033.924,-49.552,416.448,168.223,40.353,157.533
C03325=1033.918,-49.801,416.460,168.220,40.354,157.533
C03326=1033.912,-50.051,416.473,168.217,40.354,157.533
C03327=1033.906,-50.301,416.485,168.215,40.355,157.533
C03328=1033.899,-50.550,416.497,168.212,40.355,157.533
C03329=1033.894,-50.800,416.509,168.209,40.356,157.533
C03330=1033.887,-51.049,416.521,168.207,40.357,157.533
C03331=1033.881,-51.299,416.533,168.204,40.358,157.533
C03332=1033.875,-51.548,416.547,168.201,40.359,157.534
C03333=1033.867,-51.830,416.560,168.198,40.360,157.534
C03334=1033.860,-52.112,416.573,168.195,40.361,157.534
C03335=1033.853,-52.393,416.588,168.192,40.362,157.534
C03336=1033.845,-52.674,416.601,168.190,40.363,157.534
C03337=1033.839,-52.924,416.613,168.188,40.363,157.534
C03338=1033.833,-53.174,416.625,168.185,40.364,157.534
C03339=1033.826,-53.423,416.637,168.182,40.365,157.534
C03340=1033.821,-53.672,416.649,168.179,40.366,157.534
C03341=1033.814,-53.922,416.661,168.177,40.367,157.534
C03342=1033.807,-54.172,416.673,168.174,40.367,157.534
C03343=1033.801,-54.422,416.686,168.171,40.368,157.534
C03344=1033.795,-54.671,416.698,168.169,40.369,157.534
C03345=1033.788,-54.921,416.710,168.166,40.370,157.534
C03346=1033.782,-55.171,416.722,168.163,40.371,157.534
C03347=1033.776,-55.420,416.734,168.160,40.372,157.534
C03348=1033.770,-55.670,416.745,168.159,40.372,157.534
C03349=1033.764,-55.919,416.758,168.156,40.373,157.534
C03350=1033.757,-56.169,416.770,168.153,40.374,157.534
C03351=1033.751,-56.419,416.782,168.151,40.375,157.534
C03352=1033.744,-56.668,416.794,168.148,40.376,157.534
C03353=1033.738,-56.918,416.806,168.145,40.377,157.534
C03354=1033.732,-57.167,416.818,168.142,40.377,157.534
C03355=1033.725,-57.417,416.830,168.140,40.378,157.534
C03356=1033.720,-57.667,416.841,168.137,40.379,157.534
C03357=1033.713,-57.917,416.853,168.134,40.380,157.534
C03358=1033.707,-58.166,416.865,168.133,40.381,157.534
C03359=1033.700,-58.415,416.877,168.130,40.382,157.534
C03360=1033.695,-58.665,416.890,168.127,40.383,157.535
C03361=1033.688,-58.915,416.901,168.124,40.384,157.535
C03362=1033.682,-59.165,416.913,168.122,40.384,157.535
C03363=1033.676,-59.414,416.925,168.119,40.385,157.535
C03364=1033.670,-59.663,416.937,168.116,40.386,157.535
C03365=1033.663,-59.914,416.948,168.114,40.387,157.535
C03366=1033.657,-60.163,416.960,168.111,40.388,157.535
C03367=1033.651,-60.413,416.973,168.108,40.389,157.535
C03368=1033.645,-60.662,416.984,168.106,40.390,157.535
C03369=1033.638,-60.912,416.995,168.103,40.390,157.535
C03370=1033.632,-61.162,417.007,168.101,40.391,157.535
C03371=1033.626,-61.411,417.020,168.098,40.392,157.535
C03372=1033.620,-61.660,417.032,168.096,40.393,157.535
C03373=1033.613,-61.911,417.043,168.093,40.394,157.535
C03374=1033.607,-62.161,417.055,168.090,40.395,157.535
C03375=1033.601,-62.409,417.067,168.087,40.396,157.535
C03376=1033.595,-62.660,417.078,168.085,40.397,157.535
C03377=1033.588,-62.909,417.090,168.082,40.397,157.535
C03378=1033.583,-63.158,417.102,168.079,40.398,157.535
C03379=1033.577,-63.409,417.114,168.076,40.399,157.535
C03380=1033.570,-63.658,417.126,168.075,40.400,157.535
C03381=1033.564,-63.908,417.136,168.072,40.401,157.535
C03382=1033.559,-64.158,417.149,168.069,40.402,157.535
C03383=1033.552,-64.407,417.161,168.066,40.403,157.535
C03384=1033.546,-64.657,417.172,168.064,40.403,157.535
C03385=1033.539,-64.906,417.184,168.061,40.404,157.535
C03386=1033.534,-65.157,417.196,168.058,40.405,157.535
C03387=1033.528,-65.406,417.207,168.056,40.406,157.535
C03388=1033.521,-65.655,417.219,168.053,40.407,157.535
C03389=1033.515,-65.905,417.230,168.050,40.407,157.535
C03390=1033.509,-66.154,417.242,168.047,40.408,157.536
C03391=1033.503,-66.405,417.254,168.046,40.409,157.536
C03392=1033.497,-66.654,417.265,168.043,40.410,157.536
C03393=1033.491,-66.904,417.277,168.040,40.411,157.536
C03394=1033.485,-67.153,417.288,168.037,40.412,157.536
C03395=1033.479,-67.403,417.300,168.035,40.412,157.536
C03396=1033.473,-67.653,417.312,168.032,40.413,157.536
C03397=1033.466,-67.935,417.325,168.029,40.414,157.536
C03398=1033.459,-68.218,417.338,168.026,40.415,157.536
C03399=1033.452,-68.501,417.351,168.023,40.416,157.536
C03400=1033.446,-68.783,417.364,168.019,40.417,157.536
C03401=1033.439,-69.033,417.376,168.018,40.418,157.536
C03402=1033.433,-69.282,417.387,168.015,40.419,157.536
C03403=1033.427,-69.533,417.398,168.012,40.420,157.536
C03404=1033.421,-69.781,417.410,168.009,40.421,157.536
C03405=1033.415,-70.032,417.422,168.007,40.422,157.536
C03406=1033.409,-70.281,417.433,168.004,40.422,157.536
C03407=1033.403,-70.531,417.444,168.001,40.423,157.536
C03408=1033.397,-70.781,417.455,167.998,40.424,157.536
C03409=1033.390,-71.030,417.467,167.996,40.425,157.536
C03410=1033.385,-71.280,417.479,167.993,40.426,157.536
C03411=1033.379,-71.529,417.491,167.990,40.427,157.536
C03412=1033.373,-71.779,417.502,167.988,40.428,157.536
C03413=1033.367,-72.029,417.513,167.986,40.429,157.536
C03414=1033.361,-72.278,417.524,167.983,40.430,157.536
C03415=1033.355,-72.529,417.536,167.980,40.430,157.536
C03416=1033.349,-72.778,417.547,167.977,40.431,157.536
C03417=1033.343,-73.027,417.559,167.975,40.432,157.536
C03418=1033.337,-73.277,417.570,167.972,40.433,157.536
C03419=1033.331,-73.527,417.581,167.969,40.434,157.536
C03420=1033.325,-73.777,417.592,167.966,40.435,157.537
C03421=1033.320,-74.026,417.604,167.964,40.436,157.537
C03422=1033.313,-74.276,417.616,167.962,40.437,157.537
C03423=1033.307,-74.525,417.626,167.959,40.438,157.537
C03424=1033.300,-74.776,417.637,167.956,40.439,157.537
C03425=1033.294,-75.024,417.649,167.953,40.440,157.537
C03426=1033.288,-75.275,417.660,167.951,40.441,157.537
C03427=1033.282,-75.524,417.671,167.948,40.441,157.537
C03428=1033.276,-75.774,417.682,167.945,40.442,157.537
C03429=1033.270,-76.024,417.693,167.942,40.443,157.537
C03430=1033.264,-76.273,417.704,167.939,40.444,157.537
C03431=1033.258,-76.523,417.715,167.937,40.446,157.537
C03432=1033.252,-76.772,417.727,167.935,40.447,157.537
C03433=1033.246,-77.022,417.738,167.932,40.448,157.537
C03434=1033.239,-77.272,417.748,167.929,40.449,157.537
C03435=1033.233,-77.521,417.759,167.926,40.450,157.537
C03436=1033.227,-77.771,417.770,167.923,40.451,157.537
C03437=1033.221,-78.021,417.781,167.920,40.452,157.537
C03438=1033.215,-78.271,417.792,167.918,40.453,157.537
C03439=1033.209,-78.521,417.803,167.916,40.454,157.537
C03440=1033.204,-78.770,417.814,167.913,40.455,157.538
C03441=1033.197,-79.020,417.825,167.910,40.456,157.538
C03442=1033.191,-79.270,417.836,167.907,40.457,157.538
C03443=1033.185,-79.519,417.847,167.905,40.458,157.538
C03444=1033.179,-79.769,417.858,167.902,40.459,157.538
C03445=1033.173,-80.019,417.869,167.899,40.460,157.538
C03446=1033.167,-80.269,417.880,167.896,40.461,157.538
C03447=1033.160,-80.518,417.890,167.894,40.462,157.538
C03448=1033.154,-80.767,417.901,167.891,40.464,157.538
C03449=1033.148,-81.018,417.912,167.888,40.465,157.538
C03450=1033.142,-81.267,417.923,167.885,40.466,157.538
C03451=1033.136,-81.516,417.933,167.883,40.467,157.538
C03452=1033.129,-81.766,417.945,167.880,40.468,157.538
C03453=1033.123,-82.016,417.955,167.877,40.469,157.538
C03454=1033.117,-82.265,417.966,167.875,40.470,157.538
C03455=1033.110,-82.516,417.976,167.872,40.472,157.539
C03456=1033.105,-82.765,417.987,167.869,40.473,157.539
C03457=1033.099,-83.015,417.998,167.866,40.474,157.539
C03458=1033.092,-83.264,418.008,167.863,40.475,157.539
C03459=1033.086,-83.514,418.019,167.861,40.476,157.539
C03460=1033.080,-83.763,418.030,167.859,40.477,157.539
C03461=1033.073,-84.049,418.042,167.855,40.479,157.539
C03462=1033.066,-84.333,418.054,167.852,40.480,157.539
C03463=1033.059,-84.618,418.066,167.849,40.481,157.539
C03464=1033.052,-84.903,418.078,167.845,40.483,157.539
C03465=1033.046,-85.153,418.089,167.843,40.483,157.539
C03466=1033.040,-85.402,418.100,167.840,40.484,157.539
C03467=1033.034,-85.652,418.109,167.838,40.486,157.540
C03468=1033.028,-85.902,418.120,167.835,40.487,157.540
C03469=1033.021,-86.151,418.131,167.832,40.488,157.540
C03470=1033.015,-86.401,418.142,167.829,40.490,157.540
C03471=1033.010,-86.651,418.152,167.826,40.491,157.540
C03472=1033.003,-86.901,418.162,167.823,40.492,157.540
C03473=1032.997,-87.150,418.173,167.821,40.493,157.540
C03474=1032.991,-87.400,418.183,167.819,40.494,157.540
C03475=1032.985,-87.650,418.194,167.816,40.495,157.540
C03476=1032.979,-87.900,418.205,167.813,40.496,157.540
C03477=1032.973,-88.150,418.214,167.810,40.498,157.540
C03478=1032.967,-88.399,418.225,167.807,40.499,157.540
C03479=1032.961,-88.648,418.236,167.804,40.500,157.540
C03480=1032.955,-88.898,418.246,167.802,40.501,157.541
C03481=1032.949,-89.147,418.256,167.799,40.502,157.541
C03482=1032.942,-89.398,418.267,167.796,40.503,157.541
C03483=1032.937,-89.648,418.277,167.793,40.505,157.541
C03484=1032.930,-89.897,418.288,167.791,40.506,157.541
C03485=1032.925,-90.146,418.299,167.788,40.507,157.541
C03486=1032.918,-90.396,418.308,167.785,40.508,157.541
C03487=1032.913,-90.646,418.319,167.783,40.509,157.541
C03488=1032.906,-90.896,418.329,167.780,40.510,157.541
C03489=1032.900,-91.146,418.340,167.777,40.511,157.541
C03490=1032.894,-91.395,418.351,167.774,40.513,157.541
C03491=1032.888,-91.645,418.360,167.771,40.514,157.541
C03492=1032.883,-91.895,418.371,167.768,40.515,157.541
C03493=1032.876,-92.144,418.381,167.766,40.517,157.542
C03494=1032.871,-92.394,418.392,167.764,40.517,157.542
C03495=1032.864,-92.644,418.401,167.761,40.518,157.542
C03496=1032.859,-92.893,418.412,167.758,40.520,157.542
C03497=1032.853,-93.143,418.422,167.755,40.521,157.542
C03498=1032.846,-93.393,418.433,167.752,40.522,157.542
C03499=1032.840,-93.643,418.442,167.750,40.524,157.542
C03500=1032.834,-93.892,418.453,167.747,40.525,157.542
C03501=1032.829,-94.142,418.464,167.744,40.526,157.542
C03502=1032.822,-94.392,418.474,167.741,40.527,157.542
C03503=1032.817,-94.642,418.484,167.738,40.528,157.542
C03504=1032.810,-94.891,418.494,167.735,40.529,157.542
C03505=1032.805,-95.141,418.504,167.733,40.530,157.542
C03506=1032.799,-95.391,418.514,167.731,40.532,157.543
C03507=1032.793,-95.640,418.525,167.728,40.533,157.543
C03508=1032.787,-95.890,418.534,167.725,40.534,157.543
C03509=1032.781,-96.140,418.545,167.722,40.535,157.543
C03510=1032.775,-96.389,418.555,167.719,40.536,157.543
C03511=1032.770,-96.640,418.565,167.716,40.537,157.543
C03512=1032.763,-96.889,418.575,167.714,40.539,157.543
C03513=1032.758,-97.139,418.585,167.711,40.540,157.543
C03514=1032.751,-97.388,418.596,167.708,40.541,157.543
C03515=1032.746,-97.638,418.606,167.705,40.543,157.543
C03516=1032.740,-97.888,418.615,167.702,40.544,157.543
C03517=1032.733,-98.138,418.625,167.699,40.545,157.543
C03518=1032.728,-98.387,418.636,167.697,40.546,157.544
C03519=1032.722,-98.637,418.645,167.695,40.548,157.544
C03520=1032.715,-98.887,418.655,167.692,40.549,157.544
C03521=1032.710,-99.137,418.665,167.689,40.550,157.544
C03522=1032.703,-99.386,418.676,167.686,40.552,157.544
C03523=1032.697,-99.636,418.685,167.683,40.553,157.544
C03524=1032.691,-99.886,418.695,167.681,40.555,157.544
C03525=1032.685,-100.173,418.706,167.677,40.556,157.544
C03526=1032.678,-100.460,418.717,167.674,40.557,157.544
C03527=1032.671,-100.747,418.729,167.670,40.559,157.545
C03528=1032.664,-101.034,418.739,167.668,40.561,157.545
C03529=1032.658,-101.283,418.750,167.665,40.562,157.545
C03530=1032.652,-101.533,418.760,167.662,40.563,157.545
C03531=1032.646,-101.783,418.769,167.659,40.564,157.545
C03532=1032.640,-102.033,418.779,167.656,40.566,157.545
C03533=1032.634,-102.283,418.789,167.653,40.567,157.545
C03534=1032.628,-102.533,418.799,167.651,40.569,157.545
C03535=1032.622,-102.782,418.808,167.648,40.570,157.545
C03536=1032.615,-103.032,418.819,167.645,40.571,157.545
C03537=1032.609,-103.281,418.828,167.642,40.572,157.545
C03538=1032.604,-103.531,418.838,167.639,40.574,157.546
C03539=1032.598,-103.781,418.848,167.637,40.576,157.546
C03540=1032.592,-104.030,418.857,167.634,40.577,157.546
C03541=1032.586,-104.280,418.867,167.631,40.578,157.546
C03542=1032.580,-104.530,418.877,167.628,40.579,157.546
C03543=1032.574,-104.780,418.886,167.625,40.581,157.546
C03544=1032.568,-105.030,418.896,167.622,40.582,157.546
C03545=1032.562,-105.280,418.906,167.621,40.584,157.546
C03546=1032.556,-105.529,418.915,167.618,40.585,157.547
C03547=1032.551,-105.779,418.925,167.615,40.586,157.547
C03548=1032.545,-106.029,418.934,167.612,40.588,157.547
C03549=1032.538,-106.279,418.944,167.609,40.589,157.547
C03550=1032.532,-106.528,418.954,167.607,40.590,157.547
C03551=1032.526,-106.778,418.963,167.604,40.592,157.547
C03552=1032.521,-107.027,418.972,167.601,40.593,157.547
C03553=1032.514,-107.277,418.982,167.598,40.595,157.547
C03554=1032.509,-107.527,418.992,167.595,40.596,157.547
C03555=1032.503,-107.777,419.002,167.593,40.597,157.547
C03556=1032.497,-108.027,419.011,167.590,40.599,157.548
C03557=1032.491,-108.276,419.020,167.587,40.600,157.548
C03558=1032.485,-108.526,419.029,167.584,40.602,157.548
C03559=1032.479,-108.776,419.039,167.581,40.603,157.548
C03560=1032.473,-109.026,419.048,167.579,40.605,157.548
C03561=1032.467,-109.276,419.058,167.576,40.606,157.548
C03562=1032.461,-109.525,419.067,167.573,40.608,157.548
C03563=1032.455,-109.775,419.077,167.570,40.609,157.548
C03564=1032.449,-110.024,419.086,167.566,40.610,157.548
C03565=1032.443,-110.275,419.095,167.564,40.612,157.549
C03566=1032.437,-110.524,419.104,167.561,40.614,157.549
C03567=1032.431,-110.774,419.114,167.558,40.615,157.549
C03568=1032.425,-111.023,419.123,167.555,40.616,157.549
C03569=1032.419,-111.273,419.133,167.553,40.618,157.549
C03570=1032.414,-111.523,419.142,167.550,40.620,157.549
C03571=1032.407,-111.773,419.151,167.547,40.621,157.549
C03572=1032.401,-112.023,419.161,167.544,40.622,157.549
C03573=1032.395,-112.272,419.170,167.541,40.624,157.550
C03574=1032.390,-112.522,419.179,167.539,40.626,157.550
C03575=1032.384,-112.772,419.188,167.536,40.627,157.550
C03576=1032.377,-113.022,419.198,167.533,40.628,157.550
C03577=1032.372,-113.271,419.206,167.530,40.630,157.550
C03578=1032.366,-113.521,419.216,167.527,40.631,157.550
C03579=1032.360,-113.771,419.225,167.525,40.633,157.550
C03580=1032.354,-114.020,419.235,167.522,40.634,157.550
C03581=1032.348,-114.270,419.244,167.519,40.636,157.551
C03582=1032.342,-114.520,419.253,167.516,40.637,157.551
C03583=1032.337,-114.769,419.262,167.513,40.639,157.551
C03584=1032.331,-115.020,419.271,167.511,40.640,157.551
C03585=1032.325,-115.270,419.281,167.508,40.642,157.551
C03586=1032.319,-115.519,419.289,167.505,40.644,157.551
C03587=1032.312,-115.769,419.298,167.503,40.645,157.551
C03588=1032.306,-116.019,419.308,167.500,40.646,157.551
C03589=1032.300,-116.305,419.318,167.496,40.648,157.552
C03590=1032.293,-116.591,419.328,167.493,40.650,157.552
C03591=1032.286,-116.878,419.339,167.489,40.652,157.552
C03592=1032.280,-117.165,419.350,167.487,40.654,157.552
C03593=1032.274,-117.414,419.358,167.484,40.656,157.552
C03594=1032.267,-117.664,419.367,167.481,40.657,157.552
C03595=1032.262,-117.914,419.376,167.478,40.658,157.552
C03596=1032.256,-118.163,419.385,167.476,40.660,157.553
C03597=1032.250,-118.414,419.394,167.473,40.662,157.553
C03598=1032.245,-118.663,419.403,167.470,40.663,157.553
C03599=1032.238,-118.913,419.411,167.467,40.665,157.553
C03600=1032.232,-119.163,419.421,167.465,40.667,157.553
C03601=1032.226,-119.412,419.429,167.461,40.668,157.553
C03602=1032.220,-119.662,419.439,167.458,40.669,157.553
C03603=1032.215,-119.912,419.447,167.455,40.671,157.553
C03604=1032.208,-120.162,419.456,167.452,40.673,157.554
C03605=1032.203,-120.411,419.465,167.450,40.674,157.554
C03606=1032.197,-120.662,419.474,167.447,40.676,157.554
C03607=1032.191,-120.911,419.483,167.444,40.678,157.554
C03608=1032.186,-121.161,419.492,167.441,40.679,157.554
C03609=1032.179,-121.411,419.501,167.439,40.681,157.554
C03610=1032.173,-121.660,419.509,167.436,40.682,157.554
C03611=1032.168,-121.911,419.518,167.433,40.684,157.555
C03612=1032.162,-122.160,419.527,167.430,40.685,157.555
C03613=1032.155,-122.410,419.536,167.428,40.687,157.555
C03614=1032.150,-122.660,419.544,167.425,40.689,157.555
C03615=1032.144,-122.909,419.554,167.422,40.690,157.555
C03616=1032.139,-123.159,419.562,167.419,40.692,157.555
C03617=1032.132,-123.409,419.570,167.417,40.694,157.555
C03618=1032.126,-123.658,419.580,167.414,40.695,157.556
C03619=1032.121,-123.909,419.588,167.410,40.697,157.556
C03620=1032.115,-124.158,419.597,167.407,40.699,157.556
C03621=1032.109,-124.407,419.606,167.405,40.701,157.556
C03622=1032.103,-124.658,419.614,167.402,40.702,157.556
C03623=1032.098,-124.907,419.623,167.399,40.704,157.556
C03624=1032.091,-125.158,419.631,167.396,40.706,157.556
C03625=1032.086,-125.407,419.640,167.394,40.707,157.557
C03626=1032.079,-125.657,419.649,167.391,40.709,157.557
C03627=1032.074,-125.906,419.657,167.388,40.711,157.557
C03628=1032.068,-126.157,419.666,167.385,40.712,157.557
C03629=1032.062,-126.406,419.674,167.383,40.714,157.557
C03630=1032.056,-126.656,419.683,167.380,40.716,157.557
C03631=1032.051,-126.906,419.692,167.376,40.717,157.558
C03632=1032.045,-127.155,419.700,167.373,40.719,157.558
C03633=1032.039,-127.406,419.709,167.371,40.721,157.558
